// TwinCAT 3 PLC project STN500
// Title: STN500
// Company: Högskolan Väst
// Author: ANI
// ProgramVersion: 3.1.4022.3
// libraries:
//   Tc2_MC2, * (Beckhoff Automation GmbH)
//   Tc2_Standard, * (Beckhoff Automation GmbH)
//   Tc2_System, * (Beckhoff Automation GmbH)
//   Tc3_Module, * (Beckhoff Automation GmbH)
//   VisuDialogs, * (System)
//   VisuSymbols,3.5.10.0,System
// project tree:
//   DUTs/ AbsPosition.TcDUT, CommunicationData.TcDUT
//   / GlobalTextList.TcGTLO, PlcTask.TcTTO, Visualization Manager.TcVMO (not stored), VISU_TASK.TcTTO
//   GVLs/ GVL.TcGVL
//   POUs/ GantryPick.TcPOU, GantryLeave.TcPOU, GantryRobotMotion.TcPOU, GantryStatus.TcPOU, MAIN.TcPOU, PLC_PRG.TcPOU
//   VISUs/ GantryRobotVisu.TcVIS, Visualization.TcVIS
// real-time tasks:
//   TASK Device OPC UA Virtual Task: cycle T#200000us, priority 12, ADS port 350
//   TASK PlcTask: cycle T#5ms, priority 7, ADS port 351
//   TASK VISU_TASK: cycle T#100000us, priority 10, ADS port 352
// motion (NC):
//   TASK NC-Task 1 SAF: cycle T#2ms, priority 1, ADS port 501
//   TASK NC-Task 1 SVB: cycle T#4ms, priority 2, ADS port 511
//   AXIS Axis 1 (id 1)
//     General: UnitFlags=#x00000004
//     Dynamic: Acceleration=636.669, Deceleration=636.669, Jerk=445.433
//     Velo: Maximum=1000
//     OtherSettings: AllowMotionCmdToSlave=true
//     encoder EncType=19
//       EncPara: ScaleFactorNumerator=0.00162985, MaxCount=#xffffffff
//     drive DrvType=16
//       DrvPara: MaxCount=#xffffffff, DriveControlDWord=#x00020000
//         Analog: VeloReferenz=1000, ScaleFactorActTorque=0.1
//         TimeComp: TaskDelayCycles=1
//     controller CtrType=1
//       CtrPara: PriorControlFactor=1
//         PosDiffControl: Range=25
//         Observer: BandWidth=20
//   AXIS Axis 2 (id 2)
//     Dynamic: Acceleration=650.003, Deceleration=650.003, Jerk=444.737
//     Velo: Maximum=1000
//     OtherSettings: AllowMotionCmdToSlave=true
//     encoder EncType=19
//       EncPara: ScaleFactorNumerator=0.0005446764, MaxCount=#xffffffff
//     drive DrvType=16
//       DrvPara: MaxCount=#xffffffff, DriveControlDWord=#x00020000
//         Analog: VeloReferenz=1000, ScaleFactorActTorque=0.1
//         TimeComp: TaskDelayCycles=1
//     controller CtrType=1
//       CtrPara: PriorControlFactor=1
//         PosDiffControl: Range=25
//         Observer: BandWidth=20
//   AXIS Axis 3 (id 3)
//     Dynamic: Acceleration=630, Deceleration=630, Jerk=445.955
//     Velo: Maximum=1000
//     OtherSettings: AllowMotionCmdToSlave=true
//     encoder EncType=19
//       EncPara: ScaleFactorNumerator=0.000683214, MaxCount=#xffffffff
//     drive DrvType=16
//       DrvPara: MaxCount=#xffffffff, DriveControlDWord=#x00020000
//         Analog: VeloReferenz=1000, ScaleFactorActTorque=0.1
//         TimeComp: TaskDelayCycles=1
//     controller CtrType=1
//       CtrPara: PriorControlFactor=1
//         PosDiffControl: Range=25
//         Observer: BandWidth=20
// I/O:
//   DEVICE Device 1 (EtherCAT), AmsNetId 5.49.19.236.2.1
//     Term 1 (EK1200) PLC [EK1200-5000 EtherCAT Power supply (2A E-Bus)]
//       Term 2 (EK1110) [EK1110 EtherCAT extension]
//     Term 3 (EK1100) PLC Cabinet [EK1100 EtherCAT Coupler (2A E-Bus)]
//       Term 4 (EL1008) [EL1008 8Ch. Dig. Input 24V, 3ms]
//       Term 5 (EL1008) [EL1008 8Ch. Dig. Input 24V, 3ms]
//       Term 6 (EL2008) [EL2008 8Ch. Dig. Output 24V, 0.5A]
//       Term 7 (EL2008) [EL2008 8Ch. Dig. Output 24V, 0.5A]
//     Term 9 (EK1100) Gantry Robot Cabinet [EK1100 EtherCAT Coupler (2A E-Bus)]
//       Term 10 (EL1004) [EL1004 4Ch. Dig. Input 24V, 3ms]
//       Term 11 (EL1004) [EL1004 4Ch. Dig. Input 24V, 3ms]
//       Term 12 (EL1004) [EL1004 4Ch. Dig. Input 24V, 3ms]
//       Term 13 (EL2004) [EL2004 4Ch. Dig. Output 24V, 0.5A]
//       Term 16 (EL9011) [EL9011 End Terminal]
//     Drive X axis (MOVI-C MOVIDRIVE CiA402) [MOVI-C MOVIDRIVE CiA402]
//       modules: Module 1 (Mode of operation - CSP)
//     Drive Y Z axes (MOVI-C MOVIDRIVE CiA402) [MOVI-C MOVIDRIVE CiA402]
//       modules: Module 1 (Mode of operation - CSP), Module 3 (Mode of operation - CSP)
//   DEVICE Device 2 (OPC UA Virtual) STN100, AmsNetId 5.49.19.236.3.1
//   DEVICE Device 3 (OPC UA Virtual) STN200, AmsNetId 5.49.19.236.4.1
//   DEVICE Device 4 (OPC UA Virtual) STN300, AmsNetId 5.49.19.236.5.1
//   DEVICE Device 5 (OPC UA Virtual) STN400, AmsNetId 5.49.19.236.6.1
// variable links:
//   NC-Task 1 SAF/Axes/Axis 1 <-> Device 1 (EtherCAT)/Drive X axis (MOVI-C MOVIDRIVE CiA402)
//     Drive/Inputs/In/nDcOutputTime <-> InfoData/DcOutputShift
//     Drive/Inputs/In/nState1 <-> Module 1 (Mode of operation - CSP)/Inputs/Status word
//     Drive/Inputs/In/nState2 <-> Module 1 (Mode of operation - CSP)/Inputs/Status word @bit 8
//     Drive/Inputs/In/nState4 @bit 1 <-> WcState/InputToggle
//     Drive/Inputs/In/nState4 <-> WcState/WcState
//     Drive/Outputs/Out/nCtrl1 <-> Module 1 (Mode of operation - CSP)/Outputs/Control word
//     Drive/Outputs/Out/nCtrl2 <-> Module 1 (Mode of operation - CSP)/Outputs/Control word @bit 8
//     Drive/Outputs/Out/nDataOut1 <-> Module 1 (Mode of operation - CSP)/Outputs/Target position
//     Enc/Inputs/In/nDataIn1 <-> Module 1 (Mode of operation - CSP)/Inputs/Position actual value
//     Enc/Inputs/In/nDcInputTime <-> InfoData/DcInputShift
//     Enc/Inputs/In/nState4 @bit 1 <-> WcState/InputToggle
//     Enc/Inputs/In/nState4 <-> WcState/WcState
//   NC-Task 1 SAF/Axes/Axis 2 <-> Device 1 (EtherCAT)/Drive Y Z axes (MOVI-C MOVIDRIVE CiA402)
//     Drive/Inputs/In/nDcOutputTime <-> InfoData/DcOutputShift
//     Drive/Inputs/In/nState1 <-> Module 1 (Mode of operation - CSP)/Inputs/Status word
//     Drive/Inputs/In/nState2 <-> Module 1 (Mode of operation - CSP)/Inputs/Status word @bit 8
//     Drive/Inputs/In/nState4 @bit 1 <-> WcState/InputToggle
//     Drive/Inputs/In/nState4 <-> WcState/WcState
//     Drive/Outputs/Out/nCtrl1 <-> Module 1 (Mode of operation - CSP)/Outputs/Control word
//     Drive/Outputs/Out/nCtrl2 <-> Module 1 (Mode of operation - CSP)/Outputs/Control word @bit 8
//     Drive/Outputs/Out/nDataOut1 <-> Module 1 (Mode of operation - CSP)/Outputs/Target position
//     Enc/Inputs/In/nDataIn1 <-> Module 1 (Mode of operation - CSP)/Inputs/Position actual value
//     Enc/Inputs/In/nDcInputTime <-> InfoData/DcInputShift
//     Enc/Inputs/In/nState4 @bit 1 <-> WcState/InputToggle
//     Enc/Inputs/In/nState4 <-> WcState/WcState
//   NC-Task 1 SAF/Axes/Axis 3 <-> Device 1 (EtherCAT)/Drive Y Z axes (MOVI-C MOVIDRIVE CiA402)
//     Drive/Inputs/In/nDcOutputTime <-> InfoData/DcOutputShift
//     Drive/Inputs/In/nState1 <-> Module 3 (Mode of operation - CSP)/Inputs/Status word
//     Drive/Inputs/In/nState2 <-> Module 3 (Mode of operation - CSP)/Inputs/Status word @bit 8
//     Drive/Inputs/In/nState4 @bit 1 <-> WcState/InputToggle
//     Drive/Inputs/In/nState4 <-> WcState/WcState
//     Drive/Outputs/Out/nCtrl1 <-> Module 3 (Mode of operation - CSP)/Outputs/Control word
//     Drive/Outputs/Out/nCtrl2 <-> Module 3 (Mode of operation - CSP)/Outputs/Control word @bit 8
//     Drive/Outputs/Out/nDataOut1 <-> Module 3 (Mode of operation - CSP)/Outputs/Target position
//     Enc/Inputs/In/nDataIn1 <-> Module 3 (Mode of operation - CSP)/Inputs/Position actual value
//     Enc/Inputs/In/nDataIn6 @bit 1 <-> WcState/InputToggle
//     Enc/Inputs/In/nDataIn6 <-> WcState/WcState
//     Enc/Inputs/In/nDcInputTime <-> InfoData/DcInputShift
//   STN500/STN500 Instance <-> Device 1 (EtherCAT)/Term 3 (EK1100) PLC Cabinet/Term 4 (EL1008)
//     PlcTask Inputs/GVL.ixBtnControlOn <-> Channel 3/Input
//     PlcTask Inputs/GVL.ixBtnProgramStart <-> Channel 4/Input
//     PlcTask Inputs/GVL.ixBtnProgramStop <-> Channel 5/Input
//     PlcTask Inputs/GVL.ixEmergencyStopOk <-> Channel 1/Input
//     PlcTask Inputs/GVL.ixLightBeamAndGatesClosed <-> Channel 2/Input
//   STN500/STN500 Instance <-> Device 1 (EtherCAT)/Term 3 (EK1100) PLC Cabinet/Term 6 (EL2008)
//     PlcTask Outputs/GVL.qxIndControlOn <-> Channel 1/Output
//     PlcTask Outputs/GVL.qxIndProgramStart <-> Channel 2/Output
//     PlcTask Outputs/GVL.qxIndProgramStop <-> Channel 3/Output
//   STN500/STN500 Instance <-> Device 1 (EtherCAT)/Term 9 (EK1100) Gantry Robot Cabinet/Term 10 (EL1004)
//     PlcTask Inputs/GVL.ixCalSwY <-> Channel 2/Input
//     PlcTask Inputs/GVL.ixLimSwYNeg <-> Channel 3/Input
//     PlcTask Inputs/GVL.ixLimSwYPos <-> Channel 1/Input
//     PlcTask Inputs/GVL.ixLimSwZPos <-> Channel 4/Input
//   STN500/STN500 Instance <-> Device 1 (EtherCAT)/Term 9 (EK1100) Gantry Robot Cabinet/Term 11 (EL1004)
//     PlcTask Inputs/GVL.ixCalSwX <-> Channel 4/Input
//     PlcTask Inputs/GVL.ixCalSwZ <-> Channel 1/Input
//     PlcTask Inputs/GVL.ixLimSwX <-> Channel 3/Input
//     PlcTask Inputs/GVL.ixLimSwZNeg <-> Channel 2/Input
//   STN500/STN500 Instance <-> Device 1 (EtherCAT)/Term 9 (EK1100) Gantry Robot Cabinet/Term 13 (EL2004)
//     PlcTask Outputs/GVL.qxEnableSEWdrives <-> Channel 2/Output
//     PlcTask Outputs/GVL.qxGripper <-> Channel 1/Output
//   STN500/STN500 Instance <-> Device 2 (OPC UA Virtual) STN100/Object1 (OPC UA Client)/PLC1/GVL/iFromSTN500ToSTN100
//     PlcTask Outputs/GVL.iFromSTN500ToSTN100 <-> Outputs/Value
//   STN500/STN500 Instance <-> Device 2 (OPC UA Virtual) STN100/Object1 (OPC UA Client)/PLC1/GVL/iToSTN500FromSTN100
//     PlcTask Inputs/GVL.iToSTN500FromSTN100 <-> Inputs/Value
//   STN500/STN500 Instance <-> Device 3 (OPC UA Virtual) STN200/Object1 (OPC UA Client)/PLC1/GVL/iFromSTN500ToSTN200
//     PlcTask Outputs/GVL.iFromSTN500ToSTN200 <-> Outputs/Value
//   STN500/STN500 Instance <-> Device 3 (OPC UA Virtual) STN200/Object1 (OPC UA Client)/PLC1/GVL/iToSTN500FromSTN200
//     PlcTask Inputs/GVL.iToSTN500FromSTN200 <-> Inputs/Value
//   STN500/STN500 Instance <-> Device 4 (OPC UA Virtual) STN300/Object1 (OPC UA Client)/PLC1/GVL/iFromSTN500ToSTN300
//     PlcTask Outputs/GVL.iFromSTN500ToSTN300 <-> Outputs/Value
//   STN500/STN500 Instance <-> Device 4 (OPC UA Virtual) STN300/Object1 (OPC UA Client)/PLC1/GVL/iToSTN500FromSTN300
//     PlcTask Inputs/GVL.iToSTN500FromSTN300 <-> Inputs/Value
//   STN500/STN500 Instance <-> Device 5 (OPC UA Virtual) STN400/Object1 (OPC UA Client)/PLC1/GVL/iFromSTN500ToSTN400
//     PlcTask Outputs/GVL.iFromSTN500ToSTN400 <-> Outputs/Value
//   STN500/STN500 Instance <-> Device 5 (OPC UA Virtual) STN400/Object1 (OPC UA Client)/PLC1/GVL/iToSTN500FromSTN400
//     PlcTask Inputs/GVL.iToSTN500FromSTN400 <-> Inputs/Value
//   STN500/STN500 Instance <-> NC-Task 1 SAF/Axes/Axis 1
//     PlcTask Inputs/GantryRobotMotion.MCXAxisRef.NcToPlc <-> Outputs/ToPlc
//     PlcTask Outputs/GantryRobotMotion.MCXAxisRef.PlcToNc <-> Inputs/FromPlc
//   STN500/STN500 Instance <-> NC-Task 1 SAF/Axes/Axis 2
//     PlcTask Inputs/GantryRobotMotion.MCYAxisRef.NcToPlc <-> Outputs/ToPlc
//     PlcTask Outputs/GantryRobotMotion.MCYAxisRef.PlcToNc <-> Inputs/FromPlc
//   STN500/STN500 Instance <-> NC-Task 1 SAF/Axes/Axis 3
//     PlcTask Inputs/GantryRobotMotion.MCZAxisRef.NcToPlc <-> Outputs/ToPlc
//     PlcTask Outputs/GantryRobotMotion.MCZAxisRef.PlcToNc <-> Inputs/FromPlc

CONFIGURATION STN500
    RESOURCE PLC ON TwinCAT3
        TASK PlcTask(INTERVAL := T#5ms, PRIORITY := 7);
        TASK VISU_TASK(INTERVAL := T#100000us, PRIORITY := 10);
        PROGRAM MAIN WITH PlcTask : MAIN;
        PROGRAM VisuElems_Visu_Prg WITH VISU_TASK : VisuElems.Visu_Prg;
    END_RESOURCE
END_CONFIGURATION

// ---- DUTs/AbsPosition.TcDUT
TYPE AbsPosition :
STRUCT
	x:LREAL;
	y:LREAL;
	z:LREAL;
END_STRUCT
END_TYPE

// ---- DUTs/CommunicationData.TcDUT
TYPE CommunicationData :
STRUCT
	PickStation:INT;
	PickPosition:INT;
	AckPickStation:INT;
	AckPickPosition:INT;
	LeaveStation:INT;
	LeavePosition:INT;
	AckLeaveStation:INT;
	AckLeavePosition:INT;
	Status: STRING;
	ManualMode: BOOL;
	Auto: BOOL;
	Paus: BOOL;
END_STRUCT
END_TYPE

// ---- GVLs/GVL.TcGVL
{attribute 'qualified_only'}
VAR_GLOBAL
			
	//OPC-UA Communication
	iToSTN500FromSTN100 AT %I*: ARRAY[1..8] OF INT;		// From STN100
	iFromSTN500ToSTN100 AT %Q*: ARRAY[1..8] OF INT;		// To STN100

	iToSTN500FromSTN200 AT %I*: ARRAY[1..8] OF INT;		// From STN200
	iFromSTN500ToSTN200 AT %Q*: ARRAY[1..8] OF INT;		// To STN200

	iToSTN500FromSTN300 AT %I*: ARRAY[1..8] OF INT;		// From STN300
	iFromSTN500ToSTN300 AT %Q*: ARRAY[1..8] OF INT;		// To STN300

	
	iToSTN500FromSTN400 AT %I*: ARRAY[1..8] OF INT;		// From STN300
	iFromSTN500ToSTN400 AT %Q*: ARRAY[1..8] OF INT;		// To STN300
	

	//Digital I/O Gantry Robot	
	ixEmergencyStopOk		 	AT %I* 	: BOOL;			//Emergency stop reseted
	ixLightBeamAndGatesClosed 	AT %I* 	: BOOL;			//Gate closed and reseted
	ixBtnControlOn				AT %I*	: BOOL; 		//Button "Drift Till"
	ixBtnProgramStart			AT %I*	: BOOL;			//Button "Program Start"
	ixBtnProgramStop			AT %I*	: BOOL;			//Button "Program Stopp"

	ixLimSwYPos					AT %I*	: BOOL;			//End limit switches and calibration sensors
	ixCalSwY					AT %I*	: BOOL;
	ixLimSwYNeg					AT %I*	: BOOL;
	ixLimSwZPos					AT %I*	: BOOL;
	ixCalSwZ					AT %I*	: BOOL;
	ixLimSwZNeg					AT %I*	: BOOL;
	ixLimSwX					AT %I*	: BOOL;
	ixCalSwX					AT %I*	: BOOL;
	
	
	qxIndControlOn				AT %Q*	: BOOL; 		//Indication Lamp "Drift Till"
	qxIndProgramStart			AT %Q*	: BOOL;			//Indication Lamp Button "Program Start"
	qxIndProgramStop			AT %Q*	: BOOL;			//Indication Lamp Button "Program Stopp"

	qxGripper					AT %Q*	: BOOL;   		//Gripper pallets gantry robot
	qxEnableSEWdrives			AT %Q*  : BOOL;			//Enable motors XYZ axes
	
	ComData: CommunicationData;
	
END_VAR

// ---- POUs/MAIN.TcPOU
PROGRAM MAIN
VAR

END_VAR


GantryRobotMotion();
PLC_PRG();

END_PROGRAM

// ---- POUs/GantryRobotMotion.TcPOU
PROGRAM GantryRobotMotion
VAR
	
	//Speed settings Adjustible from Visu
	MCJogVelocity		: LREAL := 100.0;
	MCAutoVelocity		: LREAL := 250.0;
	mxMCButtonManLowVelocity 	: BOOL;
	

	//Homing motion Settings
	MCHomingMode	: MC_HomingMode := MC_HomingMode.MC_DefaultHoming ;
	iMCXCaibratePos 	: INT := 8;
	iMCYCaibratePos 	: INT := 8;
	iMCZCaibratePos 	: INT := 8;

	//Manual motion Settings
	MCJogMode		: E_JogMode 	:= E_JogMode.MC_JOGMODE_CONTINOUS;
	MCJogAcceleration	: LREAL := 500.0;
	MCJogDeceleration	: LREAL := 1500.0;
	MCJogJerk			: LREAL := 800.0;
	
	//Auto Motion Settings
	MCAutoAcceleration	: LREAL := 500.0;
	MCAutoDeceleration	: LREAL := 500.0;
	MCAutoJerk			: LREAL := 500.0;
	
	
	//Safe Transport Position
	MCYSafePos : LREAL := 160.0;
	MCZLiftDist : LREAL := 50.0;


	//Connection NC to Physical Servo Drives
	MCXAxisRef: AXIS_REF;
	MCYAxisRef: AXIS_REF;
	MCZAxisRef: AXIS_REF;

	
	// Auto motion Settings
	MCBufferMode   	: MC_BufferMode := MC_BufferMode.MC_Aborting;	
	
	

	//General Condition flags
	mxGeneralCOntrolOk: BOOL;
	mxButtonGeneralControlOn: BOOL;
	mxButtonGeneralControlOff: BOOL;
	mxButtonStartAuto : BOOL;
	mxButtonStopAuto : BOOL;
	mxButtonAutoMode: BOOL;
	mxGeneralControlOn: BOOL;	
	mxManualMode: BOOL;	
	mxAutoMode: BOOL;
	mxLimSwOK: BOOL;
	mxMCPowerOn: BOOL;
	mxAxesStatusOk: BOOL;
	mxAutoOn: BOOL;
	fbTONpuls1: TON;
	fbTONpuls2: TON;
	mxControlOff: BOOL;
	
	//Motor Control Function Block
	//MC  Power
	fbMCXPower: MC_Power;	//X-Axis
	mxMCXButtonByPass: BOOL;
	mxMCXPowerOn: BOOL;	

	fbMCYPower: MC_Power;	//Y-Axis
	mxMCYButtonByPass: BOOL;
	mxMCYPowerOn: BOOL;	
	
	fbMCZPower: MC_Power;	//Z-Axis
	mxMCZButtonByPass: BOOL;
	mxMCZPowerOn: BOOL;	
	
	
	// MC Read Status
	fbMCXReadStatus	: MC_ReadStatus;
	MCXAxisStatus	: ST_AxisStatus;
	mxMCXAxisError	: BOOL;

	fbMCYReadStatus	: MC_ReadStatus;
	MCYAxisStatus	: ST_AxisStatus;
	mxMCYAxisError	: BOOL;

	fbMCZReadStatus	: MC_ReadStatus;
	MCZAxisStatus	: ST_AxisStatus;
	mxMCZAxisError	: BOOL;

	
	// MC Read Actual Position
	fbMCXReadActualPosition: MC_ReadActualPosition;
	fbMCYReadActualPosition: MC_ReadActualPosition;
	fbMCZReadActualPosition: MC_ReadActualPosition;
	MCActualPos: AbsPosition;	
		
	//MC Reset
	fbMCXReset: MC_Reset;	
	fbMCYReset: MC_Reset;	
	fbMCZReset: MC_Reset;	
	mxButtonResetError:BOOL;

	//MC Homing 
	fbMCXHome: MC_Home;			//X-axis
	mxMCXButtonHoming: BOOL;
	mxMCXHomingDone: BOOL;	
	
	fbMCYHome: MC_Home;			//Y-axis
	mxMCYButtonHoming: BOOL;
	mxMCYHomingDone: BOOL;	
	
	fbMCZHome: MC_Home;			//Z-axis
	mxMCZButtonHoming: BOOL;
	mxMCZHomingDone: BOOL;	
	mxHomingDone: BOOL;	
	
	//MC Jog
	fbMCXJog: MC_Jog;			//X-Axis
	mxMCXButtonJogFWD: BOOL;
	mxMCXButtonJogBWD: BOOL;
	
	fbMCYJog: MC_Jog;			//Y-Axis
	mxMCYButtonJogFWD: BOOL;
	mxMCYButtonJogBWD: BOOL;
	
	fbMCZJog: MC_Jog;			//Z-Axis
	mxMCZButtonJogFWD: BOOL;
	mxMCZButtonJogBWD: BOOL;
	
	
	//MC Move Absolute Position	(Auto Sequence)
	fbMCXMoveAbsolute: MC_MoveAbsolute;		//X-Axis
	mxMCXMoveAbs: BOOL;
	MCXMovAbsPos: LREAL;
	MCXMoveAbsVel: LREAL;
	MCXMoveAbsACC: LREAL;
	MCXMoveAbsDec: LREAL;
	MCXMoveAbsJerk: LREAL;
	mxMCXMoveAbsDone: BOOL;

	//MC Move Absolute Position
	fbMCYMoveAbsolute: MC_MoveAbsolute;  	//Y-Axis
	mxMCYMoveAbs: BOOL;
	MCYMovAbsPos: LREAL;
	MCYMoveAbsVel: LREAL;
	MCYMoveAbsACC: LREAL;
	MCYMoveAbsDec: LREAL;
	MCYMoveAbsJerk: LREAL;
	mxMCYMoveAbsDone: BOOL;
	
	fbMCXHalt: MC_Halt;
	fbMCYHalt: MC_Halt;
	fbMCZHalt: MC_Halt;
	

	//MC Move Absolute Position
	fbMCZMoveAbsolute: MC_MoveAbsolute;		//Z-Axis
	mxMCZMoveAbs: BOOL;
	MCZMovAbsPos: LREAL;
	MCZMoveAbsVel: LREAL;
	MCZMoveAbsACC: LREAL;
	MCZMoveAbsDec: LREAL;
	MCZMoveAbsJerk: LREAL;
	mxMCZMoveAbsDone: BOOL;
	
	//Modify Position
	ModPos	: AbsPosition;
	ModPosStation: INT := 1;
	ModPosLocation:INT := 1;
	mxButtonModPosExecute : BOOL;
	mxButtonSavePos : BOOL;
	fbTONButtonModPosExecute : TON;
	mxButtonReadFile: BOOL;
	mxReminderToSave : BOOL;
	
	
	// Gripper	
	mxTogleGripper : BOOL;
	fbTONGripperOn: TON;
	fbTONGripperOff: TON;	
	
	//Auto Sequence
	iSequence: INT; 
	arrAbsPosition: ARRAY[1..4, 1..9] OF AbsPosition;	//Station 100-400 Place 1 to 9
	mxButtonGoToModPos : BOOL;
	strStatusText : STRING;
	
	
	//File handling AbsPositions XYZ
	fbFileOpen    			: FB_FileOpen;
    fbFileRead              : FB_FileRead;
    fbFileWrite             : FB_FileWrite;
    fbFileClose             : FB_FileClose;    
	hFile                   : UINT   := 0;
	mxFileOpen				: BOOL;
	mxFileRead				: BOOL;	
	mxFileWrite				: BOOL;
	mxFileClose				: BOOL;
	nFileOpenMode			: DWORD;
	mxMemSavePos: BOOL;
	mxMemReadFile: BOOL;
	fbTONFileTime: TON;

END_VAR
VAR // added by the converter: edge detectors and wires of the graphical bodies
    _rt1, _rt2, _rt3, _rt4, _rt5, _rt6, _rt7 : R_TRIG;
END_VAR

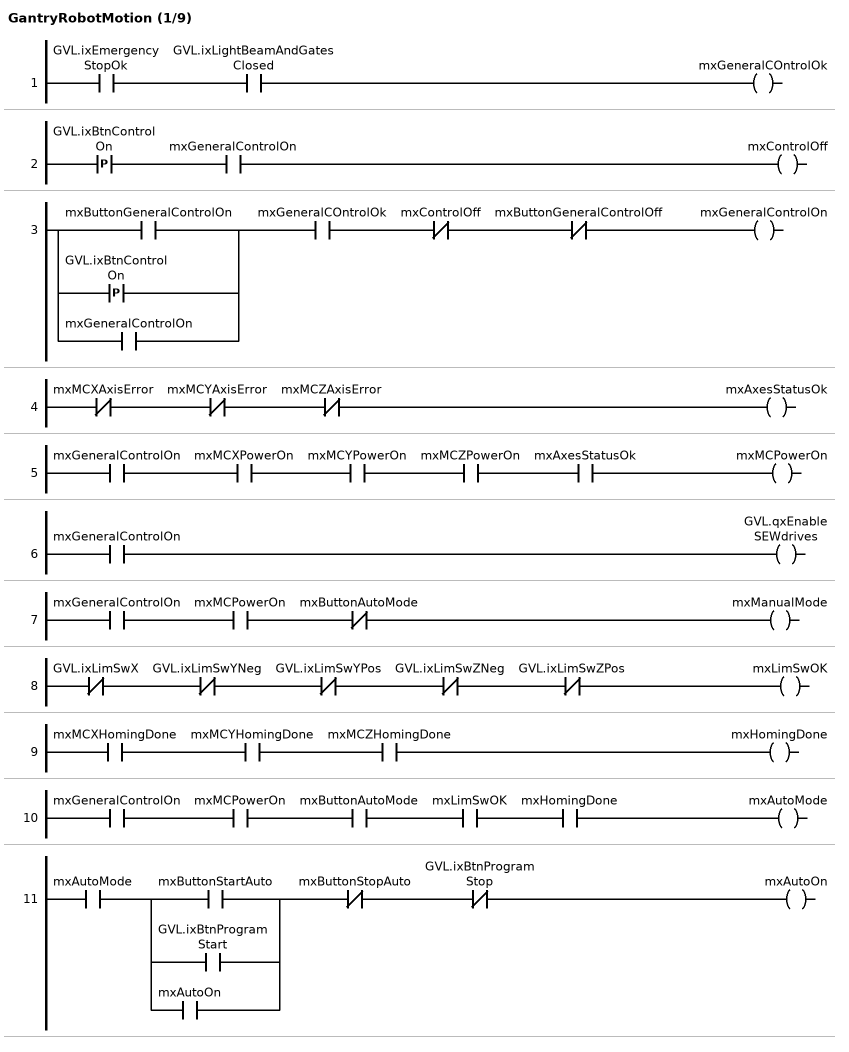
// NETWORK 1
mxGeneralCOntrolOk := GVL.ixEmergencyStopOk AND GVL.ixLightBeamAndGatesClosed;

// NETWORK 2
_rt1(CLK := GVL.ixBtnControlOn);
mxControlOff := _rt1.Q AND mxGeneralControlOn;

// NETWORK 3
_rt2(CLK := GVL.ixBtnControlOn);
mxGeneralControlOn := (mxButtonGeneralControlOn OR _rt2.Q OR mxGeneralControlOn) AND mxGeneralCOntrolOk AND NOT mxControlOff AND NOT mxButtonGeneralControlOff;

// NETWORK 4
mxAxesStatusOk := NOT mxMCXAxisError AND NOT mxMCYAxisError AND NOT mxMCZAxisError;

// NETWORK 5
mxMCPowerOn := mxGeneralControlOn AND mxMCXPowerOn AND mxMCYPowerOn AND mxMCZPowerOn AND mxAxesStatusOk;

// NETWORK 6
GVL.qxEnableSEWdrives := mxGeneralControlOn;

// NETWORK 7
mxManualMode := mxGeneralControlOn AND mxMCPowerOn AND NOT mxButtonAutoMode;

// NETWORK 8
mxLimSwOK := NOT GVL.ixLimSwX AND NOT GVL.ixLimSwYNeg AND NOT GVL.ixLimSwYPos AND NOT GVL.ixLimSwZNeg AND NOT GVL.ixLimSwZPos;

// NETWORK 9
mxHomingDone := mxMCXHomingDone AND mxMCYHomingDone AND mxMCZHomingDone;

// NETWORK 10
mxAutoMode := mxGeneralControlOn AND mxMCPowerOn AND mxButtonAutoMode AND mxLimSwOK AND mxHomingDone;

// NETWORK 11
mxAutoOn := mxAutoMode AND (mxButtonStartAuto OR GVL.ixBtnProgramStart OR mxAutoOn) AND NOT mxButtonStopAuto AND NOT GVL.ixBtnProgramStop;

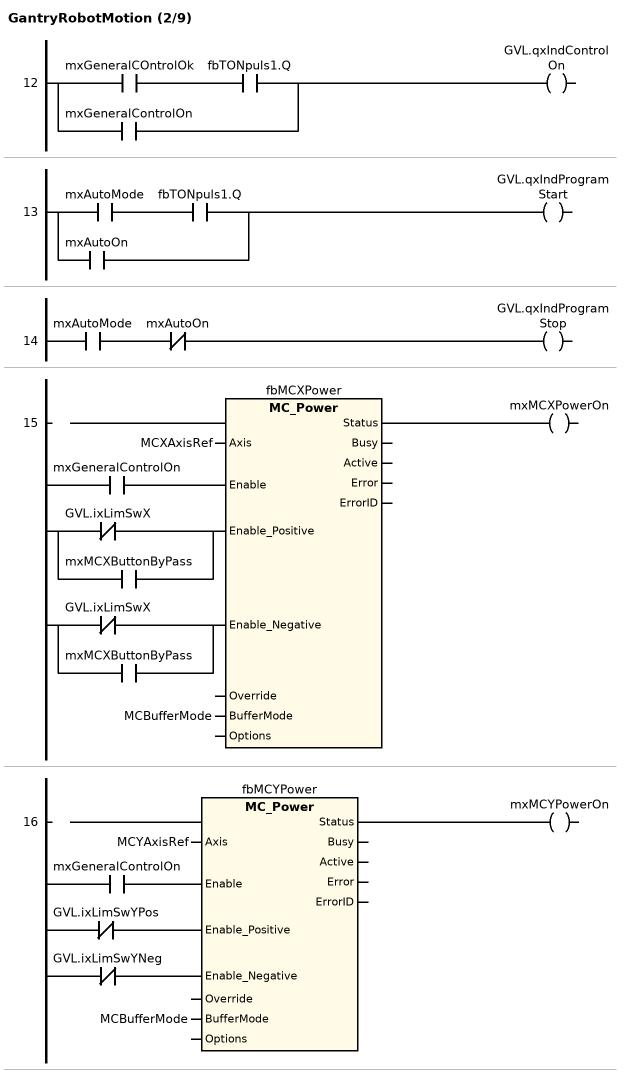
// NETWORK 12
GVL.qxIndControlOn := mxGeneralCOntrolOk AND fbTONpuls1.Q OR mxGeneralControlOn;

// NETWORK 13
GVL.qxIndProgramStart := mxAutoMode AND fbTONpuls1.Q OR mxAutoOn;

// NETWORK 14
GVL.qxIndProgramStop := mxAutoMode AND NOT mxAutoOn;

// NETWORK 15
fbMCXPower(
    Axis := MCXAxisRef,
    Enable := mxGeneralControlOn,
    Enable_Positive := NOT GVL.ixLimSwX OR mxMCXButtonByPass,
    Enable_Negative := NOT GVL.ixLimSwX OR mxMCXButtonByPass,
    BufferMode := MCBufferMode); // MC_Power
mxMCXPowerOn := fbMCXPower.Status;

// NETWORK 16
fbMCYPower(
    Axis := MCYAxisRef,
    Enable := mxGeneralControlOn,
    Enable_Positive := NOT GVL.ixLimSwYPos,
    Enable_Negative := NOT GVL.ixLimSwYNeg,
    BufferMode := MCBufferMode); // MC_Power
mxMCYPowerOn := fbMCYPower.Status;

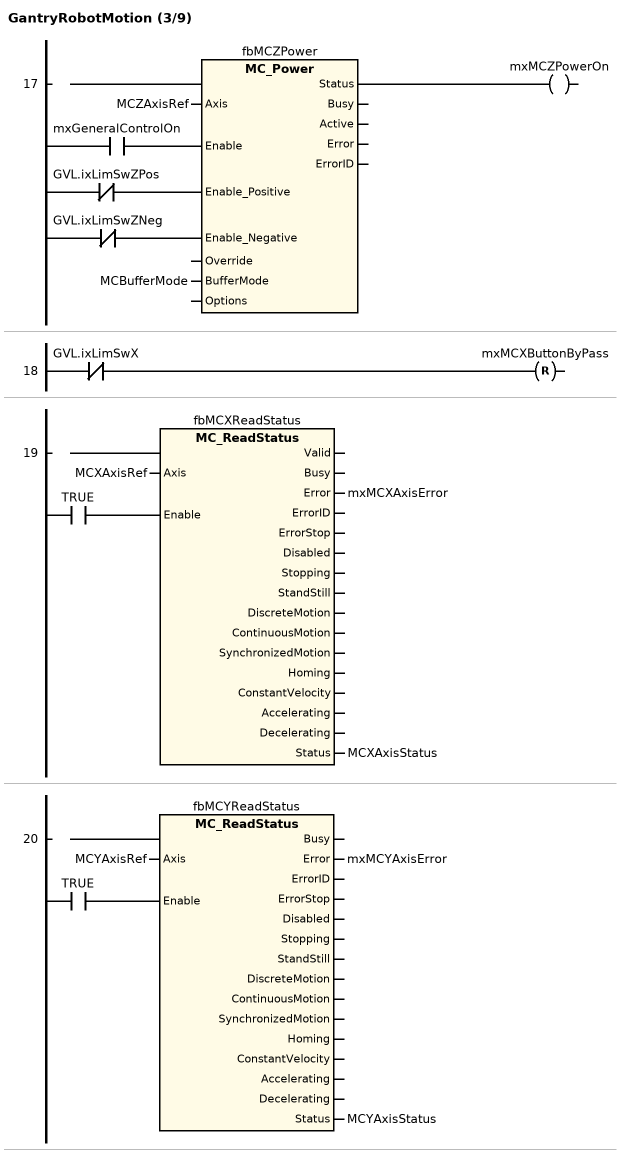
// NETWORK 17
fbMCZPower(
    Axis := MCZAxisRef,
    Enable := mxGeneralControlOn,
    Enable_Positive := NOT GVL.ixLimSwZPos,
    Enable_Negative := NOT GVL.ixLimSwZNeg,
    BufferMode := MCBufferMode); // MC_Power
mxMCZPowerOn := fbMCZPower.Status;

// NETWORK 18
mxMCXButtonByPass R= NOT GVL.ixLimSwX;

// NETWORK 19
fbMCXReadStatus(Axis := MCXAxisRef, Enable := TRUE, Error => mxMCXAxisError, Status => MCXAxisStatus); // MC_ReadStatus

// NETWORK 20
fbMCYReadStatus(Axis := MCYAxisRef, Enable := TRUE, Error => mxMCYAxisError, Status => MCYAxisStatus); // MC_ReadStatus

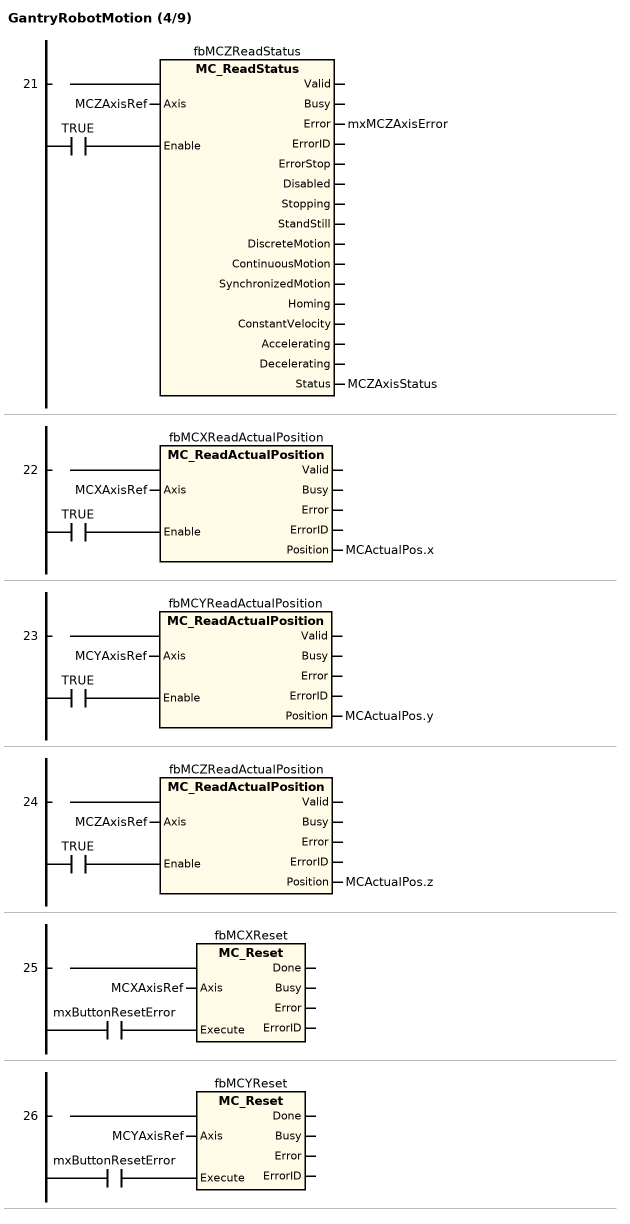
// NETWORK 21
fbMCZReadStatus(Axis := MCZAxisRef, Enable := TRUE, Error => mxMCZAxisError, Status => MCZAxisStatus); // MC_ReadStatus

// NETWORK 22
fbMCXReadActualPosition(Axis := MCXAxisRef, Enable := TRUE, Position => MCActualPos.x); // MC_ReadActualPosition

// NETWORK 23
fbMCYReadActualPosition(Axis := MCYAxisRef, Enable := TRUE, Position => MCActualPos.y); // MC_ReadActualPosition

// NETWORK 24
fbMCZReadActualPosition(Axis := MCZAxisRef, Enable := TRUE, Position => MCActualPos.z); // MC_ReadActualPosition

// NETWORK 25
fbMCXReset(Axis := MCXAxisRef, Execute := mxButtonResetError); // MC_Reset

// NETWORK 26
fbMCYReset(Axis := MCYAxisRef, Execute := mxButtonResetError); // MC_Reset

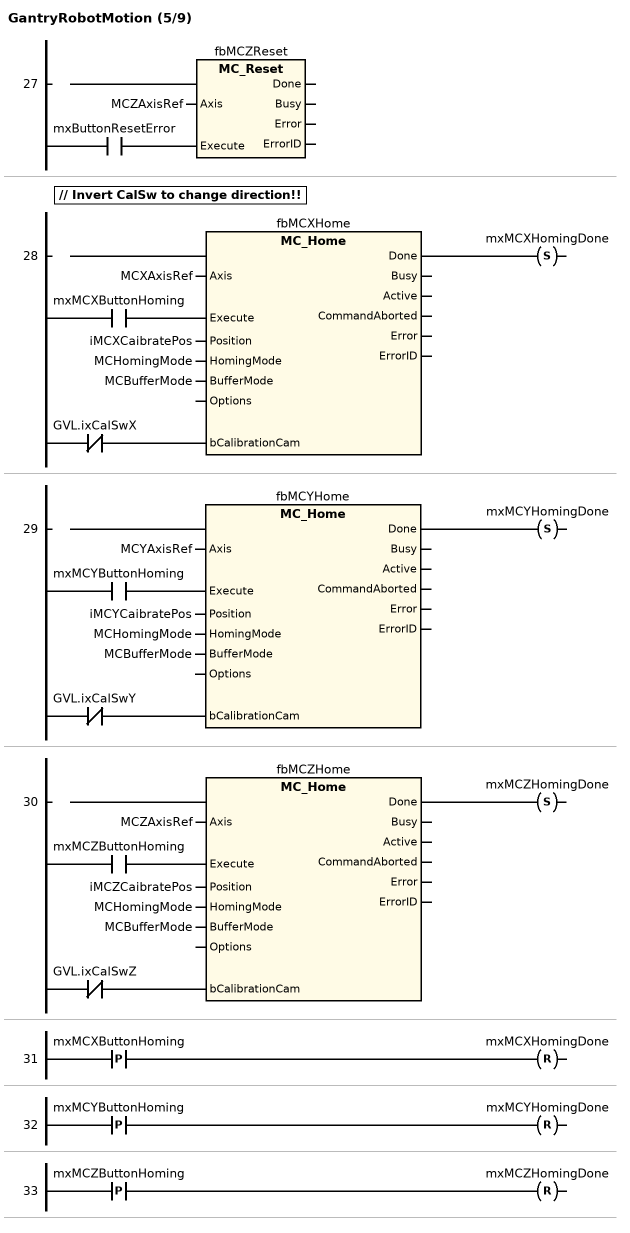
// NETWORK 27
fbMCZReset(Axis := MCZAxisRef, Execute := mxButtonResetError); // MC_Reset

// NETWORK 28
// label: // Invert CalSw to change direction!!
fbMCXHome(
    Axis := MCXAxisRef,
    Execute := mxMCXButtonHoming,
    Position := iMCXCaibratePos,
    HomingMode := MCHomingMode,
    BufferMode := MCBufferMode,
    bCalibrationCam := NOT GVL.ixCalSwX); // MC_Home
mxMCXHomingDone S= fbMCXHome.Done;

// NETWORK 29
fbMCYHome(
    Axis := MCYAxisRef,
    Execute := mxMCYButtonHoming,
    Position := iMCYCaibratePos,
    HomingMode := MCHomingMode,
    BufferMode := MCBufferMode,
    bCalibrationCam := NOT GVL.ixCalSwY); // MC_Home
mxMCYHomingDone S= fbMCYHome.Done;

// NETWORK 30
fbMCZHome(
    Axis := MCZAxisRef,
    Execute := mxMCZButtonHoming,
    Position := iMCZCaibratePos,
    HomingMode := MCHomingMode,
    BufferMode := MCBufferMode,
    bCalibrationCam := NOT GVL.ixCalSwZ); // MC_Home
mxMCZHomingDone S= fbMCZHome.Done;

// NETWORK 31
_rt3(CLK := mxMCXButtonHoming);
mxMCXHomingDone R= _rt3.Q;

// NETWORK 32
_rt4(CLK := mxMCYButtonHoming);
mxMCYHomingDone R= _rt4.Q;

// NETWORK 33
_rt5(CLK := mxMCZButtonHoming);
mxMCZHomingDone R= _rt5.Q;

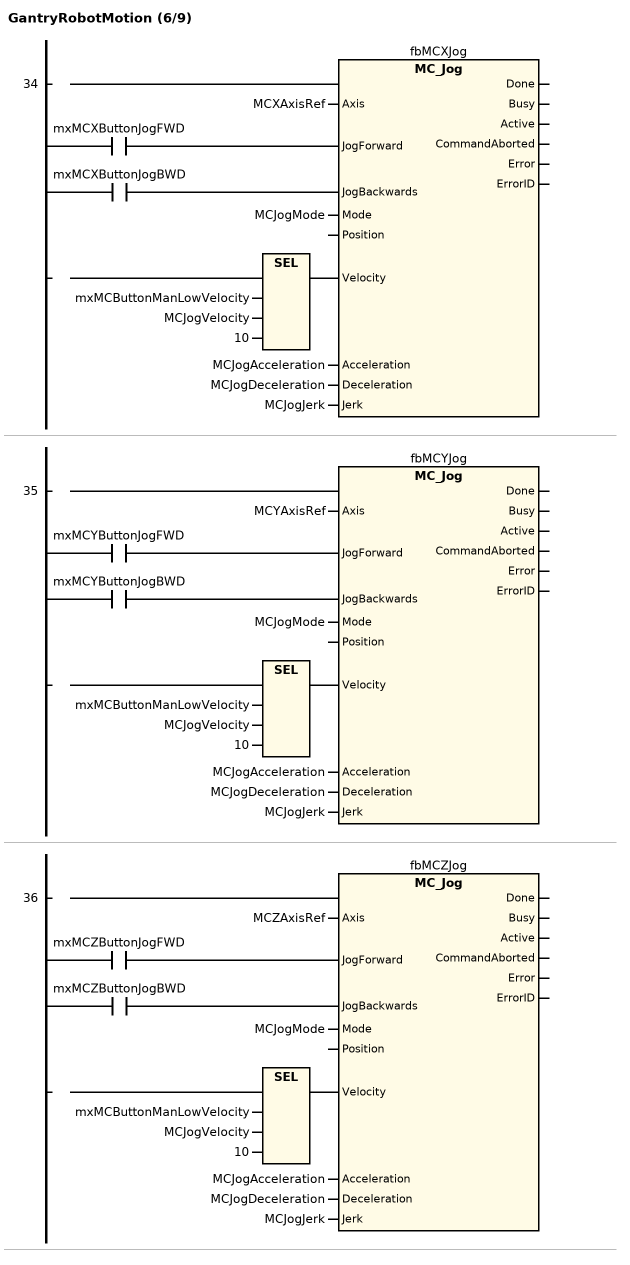
// NETWORK 34
fbMCXJog(
    Axis := MCXAxisRef,
    JogForward := mxMCXButtonJogFWD,
    JogBackwards := mxMCXButtonJogBWD,
    Mode := MCJogMode,
    Velocity := SEL(mxMCButtonManLowVelocity, MCJogVelocity, 10),
    Acceleration := MCJogAcceleration,
    Deceleration := MCJogDeceleration,
    Jerk := MCJogJerk); // MC_Jog

// NETWORK 35
fbMCYJog(
    Axis := MCYAxisRef,
    JogForward := mxMCYButtonJogFWD,
    JogBackwards := mxMCYButtonJogBWD,
    Mode := MCJogMode,
    Velocity := SEL(mxMCButtonManLowVelocity, MCJogVelocity, 10),
    Acceleration := MCJogAcceleration,
    Deceleration := MCJogDeceleration,
    Jerk := MCJogJerk); // MC_Jog

// NETWORK 36
fbMCZJog(
    Axis := MCZAxisRef,
    JogForward := mxMCZButtonJogFWD,
    JogBackwards := mxMCZButtonJogBWD,
    Mode := MCJogMode,
    Velocity := SEL(mxMCButtonManLowVelocity, MCJogVelocity, 10),
    Acceleration := MCJogAcceleration,
    Deceleration := MCJogDeceleration,
    Jerk := MCJogJerk); // MC_Jog

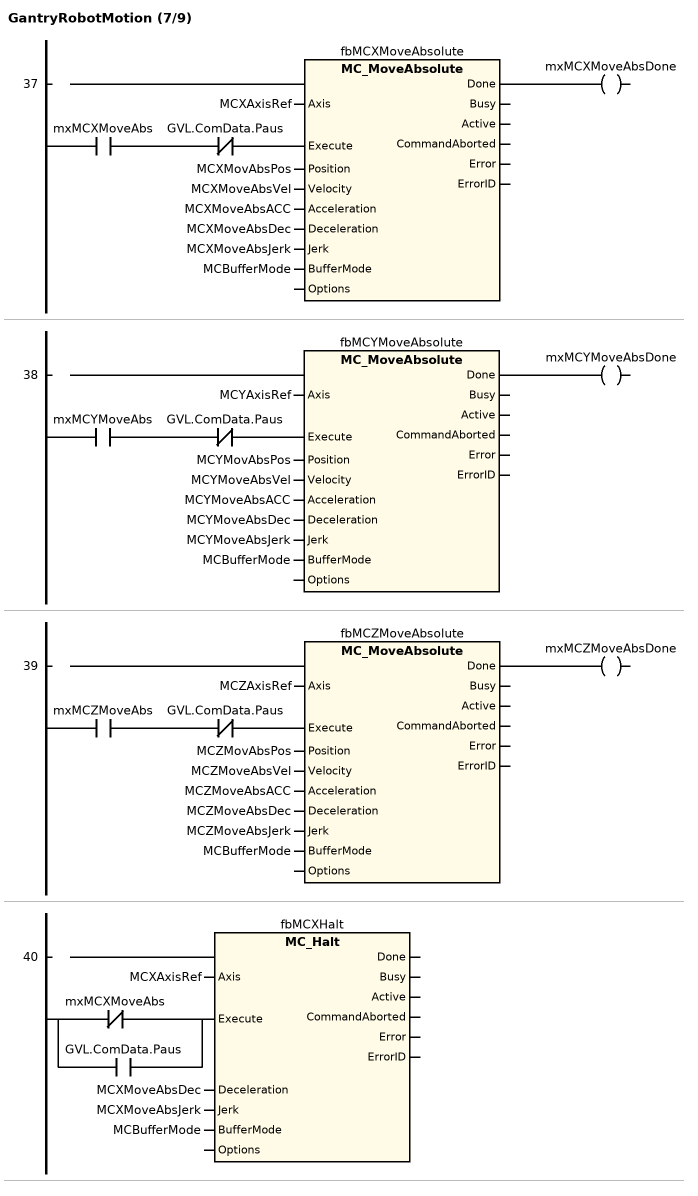
// NETWORK 37
fbMCXMoveAbsolute(
    Axis := MCXAxisRef,
    Execute := mxMCXMoveAbs AND NOT GVL.ComData.Paus,
    Position := MCXMovAbsPos,
    Velocity := MCXMoveAbsVel,
    Acceleration := MCXMoveAbsACC,
    Deceleration := MCXMoveAbsDec,
    Jerk := MCXMoveAbsJerk,
    BufferMode := MCBufferMode); // MC_MoveAbsolute
mxMCXMoveAbsDone := fbMCXMoveAbsolute.Done;

// NETWORK 38
fbMCYMoveAbsolute(
    Axis := MCYAxisRef,
    Execute := mxMCYMoveAbs AND NOT GVL.ComData.Paus,
    Position := MCYMovAbsPos,
    Velocity := MCYMoveAbsVel,
    Acceleration := MCYMoveAbsACC,
    Deceleration := MCYMoveAbsDec,
    Jerk := MCYMoveAbsJerk,
    BufferMode := MCBufferMode); // MC_MoveAbsolute
mxMCYMoveAbsDone := fbMCYMoveAbsolute.Done;

// NETWORK 39
fbMCZMoveAbsolute(
    Axis := MCZAxisRef,
    Execute := mxMCZMoveAbs AND NOT GVL.ComData.Paus,
    Position := MCZMovAbsPos,
    Velocity := MCZMoveAbsVel,
    Acceleration := MCZMoveAbsACC,
    Deceleration := MCZMoveAbsDec,
    Jerk := MCZMoveAbsJerk,
    BufferMode := MCBufferMode); // MC_MoveAbsolute
mxMCZMoveAbsDone := fbMCZMoveAbsolute.Done;

// NETWORK 40
fbMCXHalt(
    Axis := MCXAxisRef,
    Execute := NOT mxMCXMoveAbs OR GVL.ComData.Paus,
    Deceleration := MCXMoveAbsDec,
    Jerk := MCXMoveAbsJerk,
    BufferMode := MCBufferMode); // MC_Halt

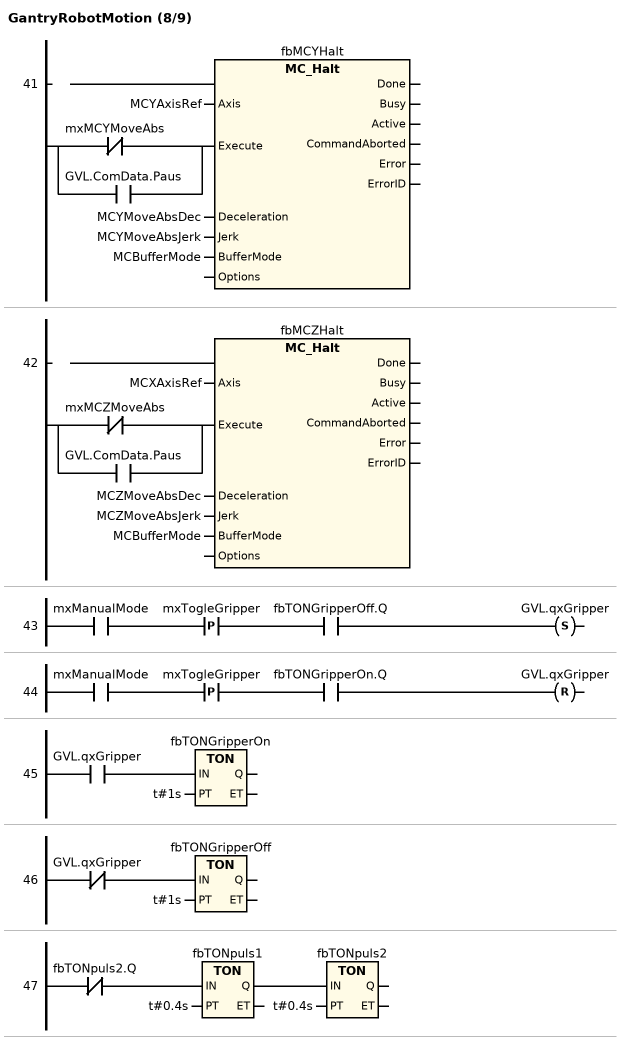
// NETWORK 41
fbMCYHalt(
    Axis := MCYAxisRef,
    Execute := NOT mxMCYMoveAbs OR GVL.ComData.Paus,
    Deceleration := MCYMoveAbsDec,
    Jerk := MCYMoveAbsJerk,
    BufferMode := MCBufferMode); // MC_Halt

// NETWORK 42
fbMCZHalt(
    Axis := MCXAxisRef,
    Execute := NOT mxMCZMoveAbs OR GVL.ComData.Paus,
    Deceleration := MCZMoveAbsDec,
    Jerk := MCZMoveAbsJerk,
    BufferMode := MCBufferMode); // MC_Halt

// NETWORK 43
_rt6(CLK := mxTogleGripper);
GVL.qxGripper S= mxManualMode AND _rt6.Q AND fbTONGripperOff.Q;

// NETWORK 44
_rt7(CLK := mxTogleGripper);
GVL.qxGripper R= mxManualMode AND _rt7.Q AND fbTONGripperOn.Q;

// NETWORK 45
fbTONGripperOn(IN := GVL.qxGripper, PT := t#1s); // TON

// NETWORK 46
fbTONGripperOff(IN := NOT GVL.qxGripper, PT := t#1s); // TON

// NETWORK 47
fbTONpuls1(IN := NOT fbTONpuls2.Q, PT := t#0.4s); // TON
fbTONpuls2(IN := fbTONpuls1.Q, PT := t#0.4s); // TON

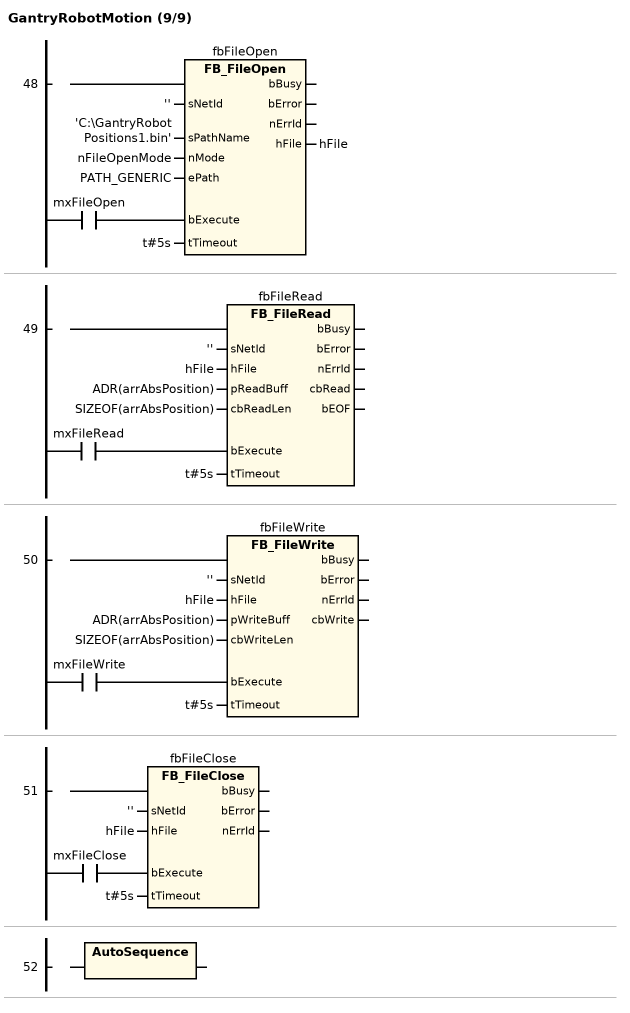
// NETWORK 48
fbFileOpen(
    sNetId := '',
    sPathName := 'C:\GantryRobotPositions1.bin',
    nMode := nFileOpenMode,
    ePath := PATH_GENERIC,
    bExecute := mxFileOpen,
    tTimeout := t#5s,
    hFile => hFile); // FB_FileOpen

// NETWORK 49
fbFileRead(
    sNetId := '',
    hFile := hFile,
    pReadBuff := ADR(arrAbsPosition),
    cbReadLen := SIZEOF(arrAbsPosition),
    bExecute := mxFileRead,
    tTimeout := t#5s); // FB_FileRead

// NETWORK 50
fbFileWrite(
    sNetId := '',
    hFile := hFile,
    pWriteBuff := ADR(arrAbsPosition),
    cbWriteLen := SIZEOF(arrAbsPosition),
    bExecute := mxFileWrite,
    tTimeout := t#5s); // FB_FileWrite

// NETWORK 51
fbFileClose(sNetId := '', hFile := hFile, bExecute := mxFileClose, tTimeout := t#5s); // FB_FileClose

// NETWORK 52
AutoSequence();

ACTION AutoSequence:


// Min Max Check Speed
IF MCJogVelocity > 250 THEN
	MCJogVelocity := 250;
END_IF
IF MCJogVelocity < 5 THEN
	MCJogVelocity := 5;
END_IF

IF MCAutoVelocity > 1000 THEN
	MCAutoVelocity := 1000;
END_IF
IF MCAutoVelocity < 100 THEN
	MCAutoVelocity := 100;
END_IF

	
// Copy status to function block interface
GVL.ComData.Status 		:= strStatusText;
GVL.ComData.ManualMode	:= mxManualMode;
GVL.ComData.Auto 		:= mxAutoOn;



CASE iSequence OF
	0:	// Init variable and read position file
		mxMCXMoveAbs := FALSE;
		mxMCYMoveAbs := FALSE;
		mxMCZMoveAbs := FALSE;
		fbTONButtonModPosExecute.PT := T#2S;
		fbTONButtonModPosExecute.IN := FALSE;
		fbTONButtonModPosExecute();

	
        // Open Gantry Robot Positions File for Read
		strStatusText := 'Reading Gantry Robot Position File'; 
		nFileOpenMode := FOPEN_MODEREAD OR FOPEN_MODEBINARY;
		mxFileOpen  := FALSE;
		mxFileRead  := FALSE;
		mxFileWrite := FALSE;
		mxFileClose := FALSE;	
		iSequence := 1;
		fbTONFileTime.IN := FALSE;
		fbTONFileTime.PT := T#3S;
		fbTONFileTime();
		
	
	1: // Wait for Opening of Gantry Robot Positions file and Check Errors
		fbTONFileTime.IN := TRUE;
		fbTONFileTime();
		mxFileOpen  := fbTONFileTime.q;
		IF mxFileOpen AND hFile > 0 AND NOT fbFileOpen.bBusy AND NOT fbFileOpen.bError THEN
			iSequence := 2;
		END_IF

	
	2:  // Read in Gantry Robot Positions File  to array of positions
		mxFileOpen  := FALSE;
		mxFileRead 	:= TRUE;
		iSequence := 3;		

			
	3:  // Wait for read Gantry Robot Positions File
		IF NOT fbFileRead.bBusy AND NOT fbFileRead.bError AND fbFileRead.cbRead = SIZEOF(arrAbsPosition) THEN
			iSequence := 4;
		END_IF
		

	4: // Close Gantry Robot Positions File
		mxFileRead  := FALSE;
		mxFileClose := TRUE;		
		strStatusText := 'Gantry Robot Position File Readed';		
		iSequence := 10;


	(* Write file *)
	5:  // Open Gantry Robot Positions Text File for Write
		strStatusText := 'Writing Gantry Robot Position File'; 
		nFileOpenMode := FOPEN_MODEWRITE OR FOPEN_MODEBINARY;
		mxFileOpen  := FALSE;
		mxFileRead  := FALSE;
		mxFileWrite := FALSE;
		mxFileClose := FALSE;	
		fbTONFileTime.IN := FALSE;
		fbTONFileTime.PT := T#3S;
		fbTONFileTime();
		iSequence := 6;
		
	
	6: // Wait for Opening of Gantry Robot Positions File and Check Errors
		fbTONFileTime.IN := TRUE;
		fbTONFileTime();
		mxFileOpen  := fbTONFileTime.Q;
		IF mxFileOpen AND hFile > 0 AND NOT fbFileOpen.bBusy AND NOT fbFileOpen.bError THEN
			iSequence := 7;
		END_IF
	
	
	7:  // Write Gantry Robot Positions File from array of positions
		mxFileOpen  := FALSE;
		mxFileWrite := TRUE;
		iSequence := 8;		

			
	8:	// Wait for Write Gantry Robot Positions File
		IF NOT fbFileWrite.bBusy AND NOT fbFileWrite.bError AND fbFileWrite.cbWrite = SIZEOF(arrAbsPosition) THEN
			iSequence := 9;
		END_IF


	9: 	// Close Gantry Robot Positions File
		strStatusText := 'Gantry Robot Positions Saved'; 		
		mxFileWrite  := FALSE;
		mxFileClose := TRUE;		
		iSequence := 10;

		
	10: // ********* Wait for auto or Modify Position, Save to file and status in Manual mode  ***************
	
		//Status text
		IF NOT GVL.ixEmergencyStopOk THEN
			strStatusText := 'Emergency Stop Activated';
		ELSIF NOT GVL.ixLightBeamAndGatesClosed THEN
			strStatusText := 'Safety Stop (Gate) Activated';
		ELSIF mxGeneralCOntrolOk AND NOT mxGeneralControlOn THEN
			strStatusText := 'Ready for General Power';
		ELSIF mxGeneralControlOn AND NOT mxMCPowerOn THEN
			strStatusText := 'Servo Drives Fault';
		ELSIF mxManualMode THEN
			strStatusText := 'Manual Mode OK';	
		ELSIF mxButtonAutoMode AND NOT mxLimSwOK THEN
			strStatusText := 'End Limit Switch Activated';
		ELSIF mxButtonAutoMode AND NOT mxHomingDone THEN
			strStatusText := 'Axes Not in reference (Run Homing)';
		ELSIF mxButtonAutoMode AND NOT mxAutoOn THEN
			strStatusText := 'Ready for Start Auto';
		ELSIF mxAutoOn THEN
			strStatusText := 'Ready for Order Auto';
		END_IF
		
					
		// Run in auto mode
		IF mxAutoOn THEN
			iSequence := 100;
		END_IF
	
		GVL.ComData.AckPickPosition := 0;
		GVL.ComData.AckPickStation := 0;
		GVL.ComData.AckLeavePosition := 0;
		GVL.ComData.AckLeaveStation := 0;
		
	
		// Move to "Modify Position" in HMI selected Robot Station and Storage Loacation 
		IF mxButtonGoToModPos AND mxManualMode AND mxHomingDone THEN //Manual Mode
			iSequence := 20;	
		END_IF
		
		// Modify position
		IF  mxButtonModPosExecute AND mxManualMode THEN
			arrAbsPosition[ModPosStation, ModPosLocation] := MCActualPos;
			mxReminderToSave := TRUE;
		END_IF
		
		// Save Position
		IF mxButtonSavePos AND NOT mxMemSavePos THEN
			iSequence := 5; //Write file
			mxReminderToSave := FALSE;
		END_IF
		mxMemSavePos := mxButtonSavePos;
		
		// Read file (UnDo)
		IF mxButtonReadFile AND NOT mxMemReadFile THEN
			iSequence := 0; //Read file
			mxReminderToSave := FALSE;
		END_IF
		mxMemReadFile := mxButtonReadFile;
		
		// Auto motion	
		IF mxAutoOn THEN
			IF GVL.ComData.LeavePosition = 0 
				AND GVL.ComData.LeaveStation = 0 
					AND GVL.ComData.PickPosition = 0 
						AND GVL.ComData.PickStation = 0 	THEN
				iSequence := 100;		//Auto mode					
			ELSE
				strStatusText := 'Clear Old Order';
			END_IF;
		END_IF
		

	
	20: 	//Init Speed Acc Dec Jerk for Manual Mode ( Goto ModPos) 
		MCXMoveAbsVel	:= MCJogVelocity ;
		MCXMoveAbsACC	:= MCJogAcceleration;
		MCXMoveAbsDec	:= MCJogDeceleration;
		MCXMoveAbsJerk	:= MCJogJerk;

		MCYMoveAbsVel	:= MCJogVelocity ;
		MCYMoveAbsACC	:= MCJogAcceleration;
		MCYMoveAbsDec	:= MCJogDeceleration;
		MCYMoveAbsJerk	:= MCJogJerk;

		MCZMoveAbsVel	:= MCJogVelocity ;
		MCZMoveAbsACC	:= MCJogAcceleration;
		MCZMoveAbsDec	:= MCJogDeceleration;
		MCZMoveAbsJerk	:= MCJogJerk;
		strStatusText := 'Moving to Modify Position';

		iSequence := 30;
		
		
	30:		// Move Y to safe position in the passage ( Goto ModPos)
		MCYMovAbsPos	:= MCYSafePos;
		mxMCYMoveAbs	:= TRUE;
		
		IF mxMCYMoveAbsDone THEN
			mxMCYMoveAbs := FALSE;
			iSequence := 40;
		END_IF
		
 		IF NOT mxButtonGoToModPos OR NOT mxManualMode THEN
			mxMCYMoveAbs:= FALSE;
			iSequence := 10;
		END_IF

		
	40:		// Move X And Z to Above Loacation ( Goto ModPos)
		MCXMovAbsPos	:= arrAbsPosition[ ModPosStation, ModPosLocation].x;
		mxMCXMoveAbs	:= TRUE;

		MCZMovAbsPos	:= arrAbsPosition[ ModPosStation, ModPosLocation].z - MCZLiftDist;
		mxMCZMoveAbs	:= TRUE;

	
		IF mxMCXMoveAbsDone AND mxMCZMoveAbsDone THEN
			mxMCXMoveAbs:= FALSE;
			mxMCZMoveAbs:= FALSE;
			iSequence 	:= 50;
		END_IF
		
		IF NOT mxButtonGoToModPos OR NOT mxManualMode THEN
			mxMCXMoveAbs:= FALSE;
			mxMCZMoveAbs:= FALSE;
			iSequence 	:= 10;
		END_IF
	
		
	50:		// Move Y in to storage ( Goto ModPos)
		MCYMovAbsPos		:= arrAbsPosition[ ModPosStation, ModPosLocation].y;
		mxMCYMoveAbs		:= TRUE;
		
		IF mxMCYMoveAbsDone THEN
			mxMCYMoveAbs 	:= FALSE;
			iSequence 		:= 60;
		END_IF
		
		IF NOT mxButtonGoToModPos OR NOT mxManualMode THEN
			mxMCYMoveAbs	:= FALSE;
			iSequence 		:= 0;
		END_IF
		
		
	60:		// Move Z down to storage ( Go to ModPos)	
		MCZMovAbsPos	:= arrAbsPosition[ ModPosStation, ModPosLocation].z;
		mxMCZMoveAbs	:= TRUE;
		
		IF mxMCYMoveAbsDone THEN
			strStatusText := 'In Modify Position';
		END_IF
		
		IF NOT mxButtonGoToModPos OR NOT mxManualMode THEN
			mxMCZMoveAbs:= FALSE;
			iSequence 	:= 10;
		END_IF

	
	
	100: 	// Init Auto speed acc and jerk ( Auto)
		MCXMoveAbsVel	:= MCAutoVelocity ;
		MCXMoveAbsACC	:= MCAutoAcceleration;
		MCXMoveAbsDec	:= MCAutoDeceleration;
		MCXMoveAbsJerk	:= MCAutoJerk;

		MCYMoveAbsVel	:= MCAutoVelocity ;
		MCYMoveAbsACC	:= MCAutoAcceleration;
		MCYMoveAbsDec	:= MCAutoDeceleration;
		MCYMoveAbsJerk	:= MCAutoJerk;

		MCZMoveAbsVel	:= MCAutoVelocity ;
		MCZMoveAbsACC	:= MCAutoAcceleration;
		MCZMoveAbsDec	:= MCAutoDeceleration;
		MCZMoveAbsJerk	:= MCAutoJerk;

		iSequence 		:= 110;

		
	110:  // Move Y to safe position in the passage ( Auto)
		MCYMovAbsPos	:= MCYSafePos;
		mxMCYMoveAbs	:= TRUE;
		strStatusText := 'Moving Y-axis to Transport Position';
	
		IF mxMCYMoveAbsDone THEN
			mxMCYMoveAbs := FALSE;
			iSequence := 120;
		END_IF
		
		IF NOT mxAutoOn THEN
			mxMCYMoveAbs:= FALSE;
			iSequence := 10;
		END_IF	

	
	120: 	// Ready for order  ( Auto)
		strStatusText := 'Ready for Order';
		iSequence := 130;

		IF NOT mxAutoOn THEN
			iSequence := 10;
		END_IF
		
		
	130:  	// *************************************** Wait for order ( Auto)  **************************************************
		IF GVL.ComData.PickPosition > 0	AND GVL.ComData.PickStation > 0 THEN
			GVL.ComData.AckPickPosition	:= 	GVL.ComData.PickPosition; //Acknowledge to function block
			GVL.ComData.AckPickStation	:= 	GVL.ComData.PickStation;
			iSequence := 200;
		END_IF		

		IF GVL.ComData.LeavePosition > 0 AND GVL.ComData.LeaveStation > 0 THEN
			GVL.ComData.AckLeavePosition	:= 	GVL.ComData.LeavePosition;
			GVL.ComData.AckLeaveStation		:= 	GVL.ComData.LeaveStation;
			iSequence := 300;
		END_IF
		

		IF NOT mxAutoOn THEN
			iSequence := 10;
		END_IF
		

	(* Auto Pickup sequence *)
	200: 	//Check Order (Auto Pickup) 	
		IF  GVL.ComData.PickPosition > 0 
			AND GVL.ComData.PickPosition <=9 
				AND GVL.ComData.PickStation > 0 
					AND GVL.ComData.PickStation <= 4 THEN
			iSequence := 210;
		ELSE
			strStatusText := 'Wrong Pickup Order Address';
			IF GVL.ComData.PickPosition = 0 AND GVL.ComData.PickStation = 0 THEN
				iSequence := 10;
			END_IF
		END_IF

		IF NOT mxAutoOn OR GVL.ComData.PickPosition = 0 OR	 GVL.ComData.PickStation = 0 THEN
			iSequence := 10;
		END_IF


	210:	// Move X And Z to Above and Outside the Loacation ( Auto Pickup)

		MCXMovAbsPos	:=  arrAbsPosition[ GVL.ComData.PickStation, GVL.ComData.PickPosition].x;
		mxMCXMoveAbs	:= TRUE;

		MCZMovAbsPos	:= arrAbsPosition[ GVL.ComData.PickStation, GVL.ComData.PickPosition].z - MCZLiftDist;
		mxMCZMoveAbs	:= TRUE;
		
		GVL.qxGripper := FALSE;
		strStatusText := 'Moving to Pickup Pallet';
		

		IF mxMCXMoveAbsDone AND mxMCZMoveAbsDone THEN
			mxMCXMoveAbs:= FALSE;
			mxMCZMoveAbs:= FALSE;
			iSequence 	:= 220;
		END_IF

		
		IF NOT mxAutoOn OR GVL.ComData.PickPosition = 0 OR	 GVL.ComData.PickStation = 0 THEN
			mxMCXMoveAbs:= FALSE;
			mxMCZMoveAbs:= FALSE;
			iSequence 	:= 10;
		END_IF
	
		
	220:	// Move Y in to storage (  Auto Pickup)
		MCYMovAbsPos		:=  arrAbsPosition[ GVL.ComData.PickStation, GVL.ComData.PickPosition].y;
		mxMCYMoveAbs		:= TRUE;
	
		IF mxMCYMoveAbsDone THEN
			mxMCYMoveAbs 	:= FALSE;
			iSequence 		:= 230;
		END_IF
		
		IF NOT mxAutoOn OR GVL.ComData.PickPosition = 0 OR	 GVL.ComData.PickStation = 0 THEN
			mxMCYMoveAbs	:= FALSE;
			iSequence 		:= 10;
		END_IF
			
		
	230:	// Move Z down to storage ( Auto Pickup)	
		MCZMovAbsPos	:= arrAbsPosition[ GVL.ComData.PickStation, GVL.ComData.PickPosition].z;
		mxMCZMoveAbs	:= TRUE;
		GVL.qxGripper := FALSE;
		
		IF mxMCZMoveAbsDone THEN
			mxMCZMoveAbs:= FALSE;
			iSequence 	:= 240;				
		END_IF
		
		IF NOT mxAutoOn OR GVL.ComData.PickPosition = 0 OR	 GVL.ComData.PickStation = 0  THEN
			mxMCZMoveAbs:= FALSE;
			iSequence 	:= 10;
		END_IF
		
	
	240:	//Grip pallet ( Auto Pickup)	
		GVL.qxGripper 	:= TRUE;
		strStatusText := 'Gripping the Pallet';
		IF fbTONGripperOn.Q THEN
			iSequence := 250;
		END_IF 
		
		IF NOT mxAutoOn OR GVL.ComData.PickPosition = 0 OR	 GVL.ComData.PickStation = 0  THEN
			iSequence 	:= 10;
		END_IF
		
		
	250: 	// Move Z up above storage ( Auto Pickup)	
		MCZMovAbsPos	:= arrAbsPosition[ GVL.ComData.PickStation, GVL.ComData.PickPosition].z - MCZLiftDist;
		mxMCZMoveAbs	:= TRUE;
		strStatusText := 'Moving out with the Pallet';
		
		IF mxMCZMoveAbsDone THEN
			mxMCZMoveAbs:= FALSE;
			iSequence := 260;
		END_IF
		
		IF NOT mxAutoOn OR GVL.ComData.PickPosition = 0 OR	 GVL.ComData.PickStation = 0  THEN
			mxMCZMoveAbs:= FALSE;
			iSequence 	:= 10;
		END_IF
		
		
	260:  	// Move Y to transport position ( Auto Pickup)	
		MCYMovAbsPos	:= MCYSafePos;
		mxMCYMoveAbs	:= TRUE;
	
		IF mxMCYMoveAbsDone THEN
			mxMCYMoveAbs := FALSE;
			GVL.ComData.AckPickPosition := 0;
			GVL.ComData.AckPickStation := 0;
			iSequence := 270;
		END_IF		
		
		IF NOT mxAutoOn OR GVL.ComData.PickPosition = 0 OR	 GVL.ComData.PickStation = 0 THEN
			mxMCYMoveAbs:= FALSE;
			iSequence := 10;
		END_IF

	
	270: 	// Wait for clear order
		strStatusText := 'Pickup pallet Done, Clear the order';
		IF 	GVL.ComData.PickStation = 0 AND GVL.ComData.PickPosition = 0 THEN
			strStatusText := 'Ready for Leave Order';
			iSequence := 130;
		END_IF	
		
		IF NOT mxAutoOn THEN
			mxMCYMoveAbs:= FALSE;
			iSequence := 10;
		END_IF

		
	300:  // Check Order 	( Auto Leave)
		IF  GVL.ComData.LeavePosition > 0 
			AND GVL.ComData.LeavePosition <=9 
				AND GVL.ComData.LeaveStation > 0 
					AND GVL.ComData.LeaveStation <= 4 THEN
			iSequence := 310;
		ELSE
			strStatusText := 'Wrong Leave Order Address';
			IF GVL.ComData.LeavePosition = 0 AND GVL.ComData.LeaveStation = 0 THEN
				iSequence := 10;
			END_IF
		END_IF

		IF NOT mxAutoOn THEN
			iSequence := 10;
		END_IF

	310:	// Move X And Z to Above and Outside the Loacation ( Auto Leave)
		MCXMovAbsPos	:= arrAbsPosition[ GVL.ComData.LeaveStation, GVL.ComData.LeavePosition].x;
		mxMCXMoveAbs	:= TRUE;

		MCZMovAbsPos	:= arrAbsPosition[ GVL.ComData.LeaveStation, GVL.ComData.LeavePosition].z - MCZLiftDist;
		mxMCZMoveAbs	:= TRUE;
		strStatusText := 'Moving to Leave Pallet';

		IF mxMCXMoveAbsDone AND mxMCZMoveAbsDone THEN
			mxMCXMoveAbs:= FALSE;
			mxMCZMoveAbs:= FALSE;
			iSequence 	:= 320;
		END_IF
		
		IF NOT mxAutoOn OR GVL.ComData.LeavePosition = 0 OR	 GVL.ComData.LeaveStation = 0 THEN
			mxMCXMoveAbs:= FALSE;
			mxMCZMoveAbs:= FALSE;
			iSequence 	:= 10;
		END_IF
	
		
	320:	// Move Y in to storage (  Auto Leave)
		MCYMovAbsPos		:= arrAbsPosition[ GVL.ComData.LeaveStation, GVL.ComData.LeavePosition].y;
		mxMCYMoveAbs		:= TRUE;
	
		IF mxMCYMoveAbsDone THEN
			mxMCYMoveAbs 	:= FALSE;
			iSequence 		:= 330;
		END_IF
		
		IF NOT mxAutoOn OR GVL.ComData.LeavePosition = 0 OR	 GVL.ComData.LeaveStation = 0 THEN
			mxMCYMoveAbs	:= FALSE;
			iSequence 		:= 10;
		END_IF
			
		
	330:	// Move Z down to storage ( Auto Leave)	
		MCZMovAbsPos	:= arrAbsPosition[ GVL.ComData.LeaveStation, GVL.ComData.LeavePosition].z;
		mxMCZMoveAbs	:= TRUE;
		
		IF mxMCZMoveAbsDone THEN
			mxMCZMoveAbs:= FALSE;
			iSequence 	:= 340;				
		END_IF
		
		IF NOT mxAutoOn OR GVL.ComData.LeavePosition = 0 OR	 GVL.ComData.LeaveStation = 0  THEN
			mxMCZMoveAbs:= FALSE;
			iSequence 	:= 10;
		END_IF
		
		
	340: 	// Release Gripper ( Auto Leave)
		GVL.qxGripper 	:= FALSE;
		strStatusText := 'Ungriping the Pallet';
		IF fbTONGripperOff.Q THEN
			iSequence := 350;
		END_IF 
		
		IF NOT mxAutoOn OR GVL.ComData.LeavePosition = 0 OR	 GVL.ComData.LeaveStation = 0  THEN
			iSequence 	:= 0;
		END_IF
		
		
	350:	// Move Z up above storage ( Auto Leave)	
		MCZMovAbsPos	:= arrAbsPosition[ GVL.ComData.LeaveStation, GVL.ComData.LeavePosition].z - MCZLiftDist;
		mxMCZMoveAbs	:= TRUE;
		strStatusText := 'Moving up from storage';
		
		IF mxMCZMoveAbsDone AND fbTONGripperOff.Q THEN
			mxMCZMoveAbs := FALSE;
			iSequence 	 := 360;
		END_IF
		
		IF NOT mxAutoOn OR GVL.ComData.LeavePosition = 0 OR	 GVL.ComData.LeaveStation = 0  THEN
			mxMCZMoveAbs := FALSE;
			iSequence 	 := 10;
		END_IF
		
		
	360: 	// Move Y to transport position ( Auto Leave)	
		MCYMovAbsPos	:= MCYSafePos;
		mxMCYMoveAbs	:= TRUE;
		strStatusText 	:= 'Moving out from storage';
	
		IF mxMCYMoveAbsDone THEN
			mxMCYMoveAbs := FALSE;
			GVL.ComData.AckLeavePosition := 0;
			GVL.ComData.AckLeaveStation := 0;
			iSequence 	 := 370;
		END_IF		
		
		IF NOT mxAutoOn OR GVL.ComData.LeavePosition = 0 OR	 GVL.ComData.LeaveStation = 0 THEN
			mxMCYMoveAbs:= FALSE;
			iSequence := 10;
		END_IF

		
	370: 	// Wait for clear order
		strStatusText 	:= 'Leave pallet Done, Clear the order';
		IF 	GVL.ComData.LeaveStation = 0 AND GVL.ComData.LeavePosition = 0 THEN
			strStatusText := 'Ready for Order';
			iSequence := 130;
		END_IF	
		
		IF NOT mxAutoOn THEN
			mxMCYMoveAbs:= FALSE;
			iSequence := 10;
		END_IF

	
END_CASE
END_ACTION

END_PROGRAM

// ---- POUs/PLC_PRG.TcPOU
PROGRAM PLC_PRG
VAR
	//Visualisation 	
	mxButtonPaus	: BOOL;

	mxAuto			: BOOL;

	//Internal use
	mxStart: BOOL;
	mxDone: BOOL;
	
	//Motion Function Blocks
	fbGantryStatus: GantryStatus;

	fbGantryPick_1: GantryPick;
	fbGantryLeave_2: GantryLeave;

	nPickStation: INT := 1;
	nPickPosition: INT := 1;
	nLeaveStation: INT := 1;
	nLeavePosition: INT := 2;
END_VAR
VAR // added by the converter: edge detectors and wires of the graphical bodies
    _w1, _w2 : BOOL;
END_VAR

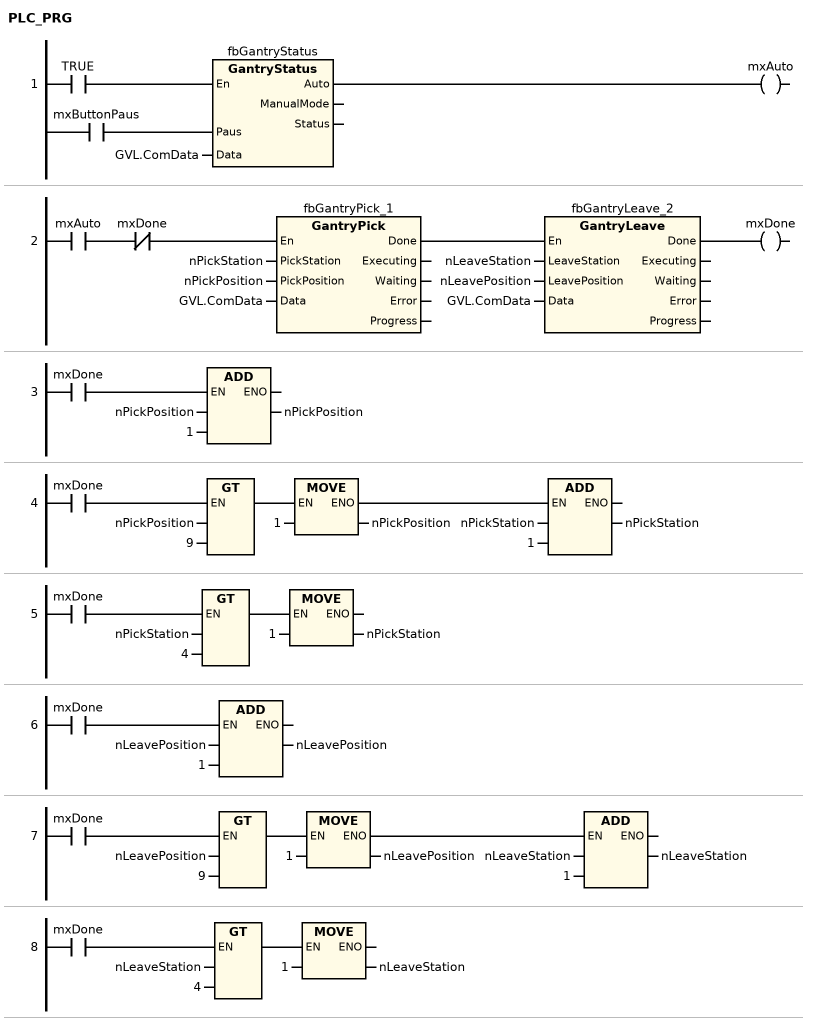
// NETWORK 1
fbGantryStatus(En := TRUE, Paus := mxButtonPaus, Data := GVL.ComData); // GantryStatus
mxAuto := fbGantryStatus.Auto;

// NETWORK 2
fbGantryPick_1(
    En := mxAuto AND NOT mxDone,
    PickStation := nPickStation,
    PickPosition := nPickPosition,
    Data := GVL.ComData); // GantryPick
fbGantryLeave_2(
    En := fbGantryPick_1.Done,
    LeaveStation := nLeaveStation,
    LeavePosition := nLeavePosition,
    Data := GVL.ComData); // GantryLeave
mxDone := fbGantryLeave_2.Done;

// NETWORK 3
IF mxDone THEN nPickPosition := nPickPosition + 1; END_IF

// NETWORK 4
_w1 := mxDone AND nPickPosition > 9;
IF _w1 THEN nPickPosition := 1; END_IF
IF _w1 THEN nPickStation := nPickStation + 1; END_IF

// NETWORK 5
IF mxDone AND nPickStation > 4 THEN nPickStation := 1; END_IF

// NETWORK 6
IF mxDone THEN nLeavePosition := nLeavePosition + 1; END_IF

// NETWORK 7
_w2 := mxDone AND nLeavePosition > 9;
IF _w2 THEN nLeavePosition := 1; END_IF
IF _w2 THEN nLeaveStation := nLeaveStation + 1; END_IF

// NETWORK 8
IF mxDone AND nLeaveStation > 4 THEN nLeaveStation := 1; END_IF

END_PROGRAM

// ---- POUs/GantryStatus.TcPOU
FUNCTION_BLOCK GantryStatus
VAR_INPUT
	En: BOOL;	
	Paus: BOOL;
END_VAR
VAR_OUTPUT
	Auto : BOOL;
	ManualMode : BOOL;	
	Status : STRING;
END_VAR
VAR_IN_OUT
	Data:CommunicationData;
END_VAR
VAR
	fbTonStartDelay: TON;
END_VAR


fbTonStartDelay( IN := Data.Auto, PT := T#1S);


Auto 		:= fbTonStartDelay.Q;
ManualMode 	:= Data.ManualMode;
Status 		:= Data.Status;
Data.Paus := Paus;

END_FUNCTION_BLOCK

// ---- POUs/GantryPick.TcPOU
FUNCTION_BLOCK GantryPick
VAR_INPUT
	En: BOOL;
	PickStation: INT;
	PickPosition: INT;
END_VAR
VAR_OUTPUT
	Done: BOOL;
	Executing: BOOL;
	Waiting: BOOL;
	Error: BOOL;
	Progress: INT;
END_VAR
VAR_IN_OUT
	Data:CommunicationData;
END_VAR
VAR
END_VAR


IF En THEN

	// Auto sequence pick pallet
	CASE Progress OF
		0:	//Clear old order
			Data.PickStation := 0;
			Data.PickPosition := 0;
			Progress := 10;

		10:	//Start gantry robot auto squence
			IF Data.Auto AND PickStation > 0 AND  PickStation <= 4 AND PickPosition > 0 AND PickPosition <= 9 THEN
				Data.PickStation := PickStation;
				Data.PickPosition := PickPosition;
				Executing := FALSE;
				Waiting := FALSE;
				Error := FALSE;
				Progress := 30;
			ELSE
				Executing := FALSE;
				Waiting := FALSE;
				Error := TRUE;
			END_IF

		30: // Check acknowledge from GantryRobot
			IF Data.AckPickStation = PickStation AND Data.AckPickPosition = PickPosition THEN
				Executing := TRUE;
				Waiting := FALSE;
				Error := FALSE;
				Progress := 50;
			ELSE
				Executing := FALSE;
				Waiting := TRUE;
				Error := NOT Data.Auto;
			END_IF
			
		50: // Wait for gantry auto squence ready and clear order	
			IF Data.AckPickStation = 0 AND Data.AckPickPosition = 0 THEN
				Data.PickStation := 0;
				Data.PickPosition := 0;
				Executing := FALSE;
				Waiting := FALSE;
				Error := FALSE;
				Progress := 100;
			ELSE
				Executing := TRUE;
				Waiting := FALSE;
				Error := NOT Data.Auto;
			END_IF
		
		100: // Operation done
			Done := TRUE;
	END_CASE

ELSE //En
	IF Progress > 0 THEN
		Data.PickStation := 0;
		Data.PickPosition := 0;	
	END_IF
	Progress := 0;
	Done := FALSE;
	Executing := FALSE;
	Waiting := FALSE;
	Error := FALSE;
END_IF

END_FUNCTION_BLOCK

// ---- POUs/GantryLeave.TcPOU
FUNCTION_BLOCK GantryLeave
VAR_INPUT
	En: BOOL;
	LeaveStation: INT;
	LeavePosition: INT;
END_VAR
VAR_OUTPUT
	Done: BOOL;
	Executing: BOOL;
	Waiting: BOOL;
	Error: BOOL;
	Progress: INT;
END_VAR
VAR_IN_OUT
	Data:CommunicationData;
END_VAR
VAR
END_VAR

IF En THEN
	
	// Auto sequence leave pallet
	CASE Progress OF
		0:	//Clear old order
			Data.LeaveStation := 0;
			Data.LeavePosition := 0;
			Progress := 10;

		10:	//Start gantry robot auto squence
			IF Data.Auto AND LeaveStation > 0 AND  LeaveStation <= 4 AND LeavePosition > 0 AND LeavePosition <= 9 THEN
				Data.LeaveStation  := LeaveStation;
				Data.LeavePosition := LeavePosition;
				Executing := FALSE;
				Waiting := FALSE;
				Error := FALSE;
				Progress := 30;
			ELSE
				Executing := FALSE;
				Waiting := FALSE;
				Error := TRUE;
			END_IF

		30: // Check acknowledge from GantryRobot
			IF Data.AckLeaveStation = LeaveStation AND Data.AckLeavePosition = LeavePosition THEN
				Executing := TRUE;
				Waiting := FALSE;
				Error := FALSE;
				Progress := 50;
			ELSE
				Executing := FALSE;
				Waiting := TRUE;
				Error := NOT Data.Auto;
			END_IF
			
		50: // Wait for gantry auto squence ready and clear order	
			IF Data.AckLeaveStation = 0 AND Data.AckLeavePosition = 0 THEN
				Data.LeaveStation := 0;
				Data.LeavePosition := 0;
				Executing := FALSE;
				Waiting := FALSE;
				Error := FALSE;
				Progress := 100;
			ELSE
				Executing := TRUE;
				Waiting := FALSE;
				Error := NOT Data.Auto;
			END_IF
		
		100: // Operation done
			Done := TRUE;
	END_CASE

ELSE //En
	IF Progress > 0 THEN
		Data.LeaveStation := 0;
		Data.LeavePosition := 0;	
	END_IF
	Progress := 0;
	Done := FALSE;
	Executing := FALSE;
	Waiting := FALSE;
	Error := FALSE;
END_IF

END_FUNCTION_BLOCK

// ---- GlobalTextList.TcGTLO
TEXTLIST GlobalTextList
  263 = ' Y-Axis %s'
  1185 = '%s'
  489 = 'ABB Go To Conveyor 1'
  490 = 'ABB Go To Conveyour 2'
  485 = 'ABB Go To Home'
  486 = 'ABB Go To Sensor'
  487 = 'ABB Go To Storage'
  488 = 'ABB Go To Table'
  986 = 'ABB PickLeave Conv. 1'
  987 = 'ABB PickLeave Conv. 2'
  983 = 'ABB PickLeave Sensor'
  984 = 'ABB PickLeave Storage'
  985 = 'ABB PickLeave Table'
  840 = 'ABB Status'
  91 = 'Actual Axes Positions'
  67 = 'Actual Position X-Axis %S'
  780 = 'Actual Position X-Axis %s'
  374 = 'Actual Position Y-Axis %s'
  492 = 'Actual Position Z-Axis %s'
  746 = 'AUTO'
  191 = 'Auto                        Manual'
  126 = 'Auto                  Manual'
  493 = 'Auto: %s'
  762 = 'Auto: %s    mm/s'
  413 = 'Auto: %s mm/s'
  269 = 'Axtual Position X %s'
  686 = 'Black Stop Button'
  694 = 'Busy'
  491 = 'By Pass'
  514 = 'By Pass \nEnd Limit X'
  336 = 'By Pass End Limit'
  214 = 'Calibrate Axes'
  695 = 'Communicator'
  965 = 'Communicator Enable'
  430 = 'Control On'
  1616 = "Don't forget to save changes!"
  1083 = "Don't forget to save!"
  998 = 'Done'
  1640 = 'Dont forget to save Positions'
  137 = 'Dont forget to save the \nPositions!'
  194 = 'Dont forget to save the Positions!'
  473 = 'Edit \nSTN100'
  458 = 'EM Stop'
  992 = 'EM Stop OK'
  724 = 'Emergency Stop'
  624 = 'Emergency Stop OK'
  505 = 'Emergency Stopop OK'
  936 = 'End Limit SW'
  66 = 'End Limit SW '
  765 = 'End Limit SW OK'
  1001 = 'Error'
  696 = 'Error %s'
  999 = 'Executing'
  997 = 'Function call'
  465 = 'Gantry Leave'
  464 = 'Gantry Pick'
  81 = 'Gantry Robot'
  441 = 'Gantry Robot\nMenu'
  566 = 'Gate '
  402 = 'Gate Closed'
  571 = 'Gate Closed and Reset'
  567 = 'Gate Closed and reseted'
  1091 = 'Gate Closed and Reseted'
  788 = 'Gate Closed Reset'
  43 = 'Gate OK '
  109 = 'General Conditions'
  996 = 'General Control '
  210 = 'General Control \nOn'
  174 = 'General Control On'
  60 = 'General Power\nOff'
  708 = 'General Power\nOn'
  404 = 'Go To '
  935 = 'Go To \nPosition'
  4 = 'Go To \nStorage Position'
  443 = 'Go To Storage Position'
  829 = 'Gripper'
  1144 = 'GroupBox'
  605 = 'Heart beat'
  382 = 'HOMING'
  140 = 'Homing X '
  133 = 'Homing Y '
  6 = 'Homing Z'
  543 = 'Light Beam'
  1111 = 'Location: %4.1f'
  729 = 'Location: %S'
  544 = 'Location: %s'
  223 = 'Main Menu'
  74 = 'Manual              Auto'
  621 = 'Manual        Auto'
  468 = 'Manual      Auto'
  459 = 'Manual  LOW Speed'
  595 = 'Manual Controls'
  1043 = 'Manual: %s mm/s'
  362 = 'Mod Pos '
  1483 = 'Mod Pos \n'
  1054 = 'Mod Pos \n\nSelected Location'
  665 = 'Mod Pos \n\nSelected Location'
  246 = 'Mod Pos \nSelected Location'
  692 = 'Modify Storage Position'
  842 = 'Operating mode %d'
  911 = 'Override Speed: %s'
  1219 = 'Override: %s'
  867 = 'Override: %s  %'
  1155 = 'PAUS'
  988 = 'Pick'
  1160 = 'Place'
  783 = 'Place 1'
  284 = 'Place 2'
  781 = 'Place 3'
  250 = 'Place 4'
  703 = 'Place 5'
  343 = 'Place 6'
  1179 = 'Place 7'
  247 = 'Place 8'
  480 = 'Place 9'
  989 = 'Pos\n%s'
  467 = 'Pos \n%s'
  823 = 'Position'
  1392 = 'Position %s'
  946 = 'Power\nOn'
  790 = 'Power \nOff'
  606 = 'Program number: %d'
  330 = 'Read'
  1617 = 'Reference run Axes'
  807 = 'Reset \nServo Drives'
  632 = 'Reset Servo Drives'
  604 = 'RPC Remote Procedural Call'
  603 = 'Running'
  841 = 'Running mode %d'
  1310 = 'SAve'
  1444 = 'Save'
  1220 = 'Save \nPositions!'
  297 = 'Save changes on file!'
  193 = 'Save Ented\nPosition'
  268 = 'Save Entered\nPosition'
  283 = 'Save Entred\nPosition'
  990 = 'Save or Undo changes!'
  1791 = 'Save or UnDo changes!'
  248 = 'Save or UnDo the changes!'
  612 = 'Save or Undo yhe changes!'
  560 = 'Save or UnDo yhe changes!'
  19 = 'Speed Settings'
  101 = 'Start Auto'
  466 = 'Station\n%s'
  945 = 'Station address \n%s'
  396 = 'Station: %S'
  586 = 'Station: %s'
  1075 = 'Status: %s'
  707 = 'STN100'
  226 = 'STN200'
  377 = 'STN300'
  63 = 'STN400'
  625 = 'STN500'
  323 = 'Stop Auto'
  524 = 'Stop Button'
  152 = 'Stop Button (Black)'
  674 = 'Stop Button (Black) OK'
  527 = 'UnDo'
  1089 = 'UnDo Entered'
  363 = 'UnDo Entered \nPosition'
  813 = 'Undo Entered \nPosition'
  1000 = 'Waiting'
  714 = 'X'
  333 = 'X '
  859 = 'X                  Y                Z\nReset\nServo Drives'
  153 = 'X                 Y               Z\nReset\nServo Drives'
  141 = 'X                Y                Z\nReset\nServo Drives'
  436 = 'X                Y               Z\nReset\nServo Drives'
  180 = 'X              Y            Z\nReset\nServo Drives'
  228 = 'X              Y            Z\nReset \nServo Drives'
  327 = 'X              Y            Z\nReset Error\nServo Drives'
  855 = 'X      Y     Z\nReset \nServo Drives'
  289 = 'X +'
  412 = 'X-'
  115 = 'X-Axis %s'
  910 = 'X: %4.1f'
  875 = 'X: %f4.1'
  457 = 'X: %S'
  824 = 'X: %s'
  381 = 'Y'
  482 = 'Y+'
  668 = 'Y-'
  142 = 'Y-Axis %s'
  754 = 'Y: %4.1f'
  879 = 'Y: %f4.1'
  1038 = 'Y: %S'
  245 = 'Y: %s'
  38 = 'z'
  406 = 'Z'
  832 = 'z+'
  975 = 'z-'
  348 = 'Z-Axis %s'
  1274 = 'Z: %4.1f'
  789 = 'Z: %f4.1'
  192 = 'Z: %S'
  655 = 'Z: %s'
END_TEXTLIST

// ---- VISUs/GantryRobotVisu.TcVIS
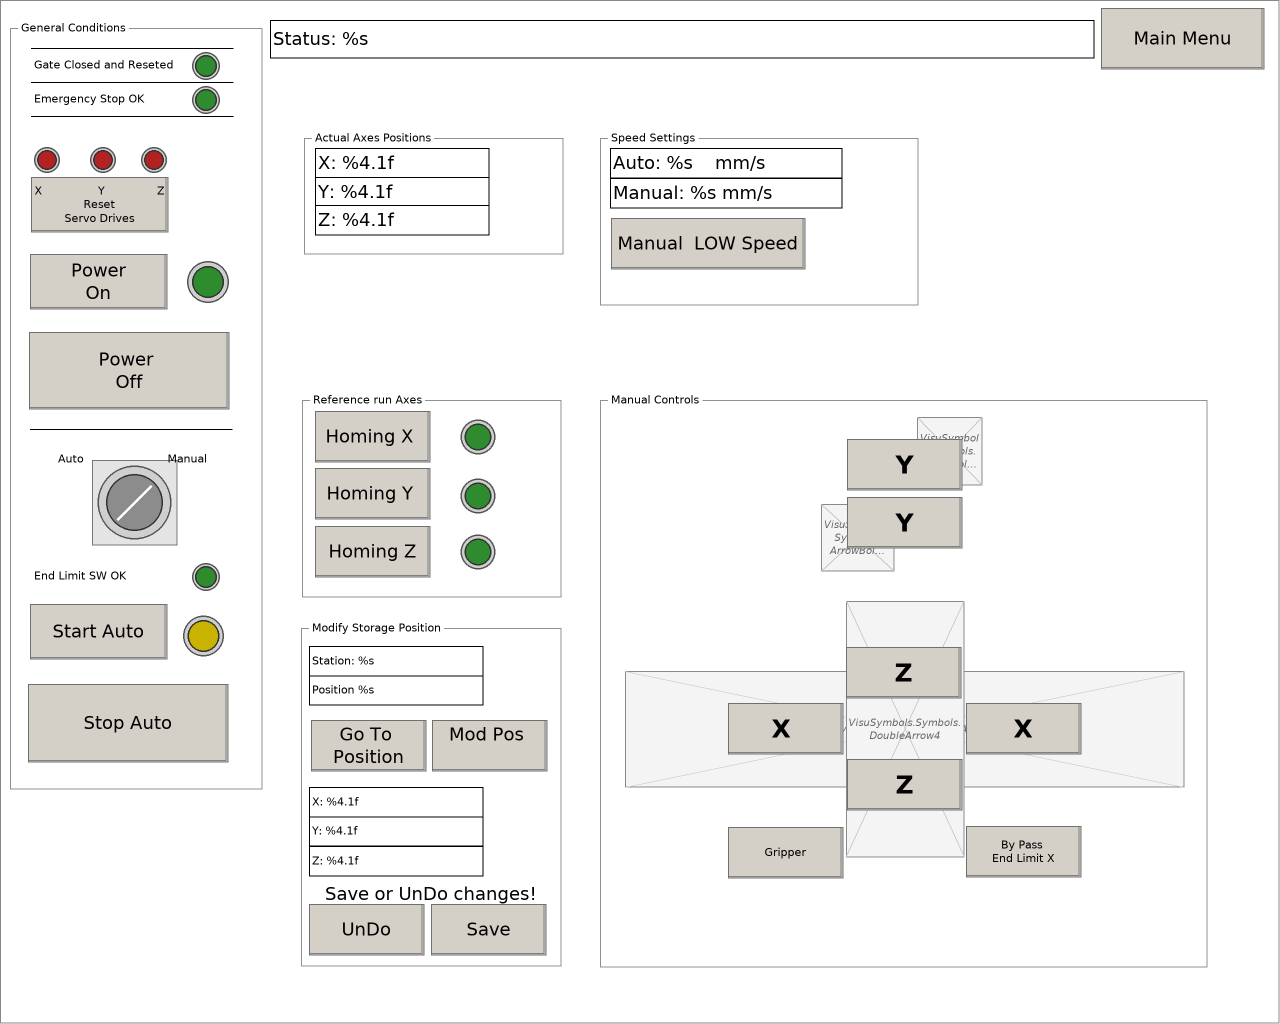
VISUALIZATION GantryRobotVisu  // 1280x1024
    GroupBox (600,392 607x575), "Manual Controls"
        Image (221,112 73x67), image: VisuSymbols.Symbols.ArrowBoldLeftDown
        Image (317,25 65x68), image: VisuSymbols.Symbols.ArrowBoldRightUp
        Image (25,279 559x116), image: VisuSymbols.Symbols.DoubleArrow3
        Image (246,209 118x256), image: VisuSymbols.Symbols.DoubleArrow4
        Button (247,105 115x51), "Y", input disabled if: NOT GantryRobotMotion.mxManualMode
            tap GantryRobotMotion.mxMCYButtonJogFWD
        Button (247,47 115x51), "Y", input disabled if: NOT GantryRobotMotion.mxManualMode
            tap GantryRobotMotion.mxMCYButtonJogBWD
        Button (128,435 115x51), "Gripper", input disabled if: NOT GantryRobotMotion.mxManualMode
            tap GantryRobotMotion.mxTogleGripper
        Button (366,434 115x51), "By Pass End Limit X", invisible if: NOT GantryRobotMotion.mxManualMode, input disabled if: NOT GVL.ixLimSwX
            toggle GantryRobotMotion.mxMCXButtonByPass
        Button (247,367 115x51), "Z", input disabled if: NOT GantryRobotMotion.mxManualMode
            tap GantryRobotMotion.mxMCZButtonJogFWD
        Button (246,255 115x51), "Z", input disabled if: NOT GantryRobotMotion.mxManualMode
            tap GantryRobotMotion.mxMCZButtonJogBWD
        Button (366,311 115x51), "X", input disabled if: NOT GantryRobotMotion.mxManualMode
            tap GantryRobotMotion.mxMCXButtonJogBWD
        Button (128,311 115x51), "X", input disabled if: NOT GantryRobotMotion.mxManualMode
            tap GantryRobotMotion.mxMCXButtonJogFWD
    GroupBox (10,20 252x769), "General Conditions"
        Button (20,234 137x55), "Power On", input disabled if: NOT GantryRobotMotion.mxGeneralCOntrolOk
            tap GantryRobotMotion.mxButtonGeneralControlOn
        Label (21,36 150x32)
        Label (21,29 160x32), "Gate Closed and Reseted"
        Lamp1 (178,30 36x32), variable: GVL.ixLightBeamAndGatesClosed, style: Lamp-Lamp1-Green
        Label (21,63 157x32), "Emergency Stop OK"
        Lamp1 (178,64 36x32), variable: GVL.ixEmergencyStopOk, style: Lamp-Lamp1-Green
        Lamp1 (170,238 56x48), variable: GVL.qxIndControlOn, style: Lamp-Lamp1-Green
        Lamp1 (170,592 47x48), variable: GVL.qxIndProgramStart, style: Lamp-Lamp1-Yellow
        Label (21,540 120x32), "End Limit SW OK"
        Lamp1 (178,541 36x32), variable: GantryRobotMotion.mxLimSwOK, style: Lamp-Lamp1-Green
        Line (21,28) (223,28)
        Line (21,62) (223,62)
        Line (21,96) (223,96)
        RotarySwitch (75,440 99x85), variable: GantryRobotMotion.mxButtonAutoMode, behaviour: TOGGLE, style: Switch-RotarySwitch-Gray
        Label (26,423 193x32), "Auto Manual"
        Line (20,409) (222,409)
        Button (20,584 137x55), "Start Auto", input disabled if: NOT GantryRobotMotion.mxAutoMode
            tap GantryRobotMotion.mxButtonStartAuto
        Lamp1 (128,125 32x30), variable: GantryRobotMotion.mxMCXAxisError, style: Lamp-Lamp1-Red
        Lamp1 (77,125 32x30), variable: GantryRobotMotion.mxMCXAxisError, style: Lamp-Lamp1-Red
        Lamp1 (21,125 32x30), variable: GantryRobotMotion.mxMCXAxisError, style: Lamp-Lamp1-Red
        Button (21,157 137x55), "X Y Z Reset Servo Drives"
            tap GantryRobotMotion.mxButtonResetError
        Button (19,312 200x77), "Power Off", input disabled if: NOT GantryRobotMotion.mxGeneralCOntrolOk
            tap GantryRobotMotion.mxButtonGeneralControlOff
        Button (18,664 200x78), "Stop Auto", input disabled if: NOT GantryRobotMotion.mxAutoMode
            tap GantryRobotMotion.mxButtonStopAuto
    GroupBox (304,130 259x124), "Actual Axes Positions"
        Rectangle (11,18 174x30), "X: %4.1f", text variable: GantryRobotMotion.MCActualPos.x
        Rectangle (11,47 174x30), "Y: %4.1f", text variable: GantryRobotMotion.MCActualPos.y
        Rectangle (11,75 174x30), "Z: %4.1f", text variable: GantryRobotMotion.MCActualPos.z
    Button (1101,8 163x61), "Main Menu"
        OnMouseClick: change screen: Visualization
    Rectangle (270,20 824x38), "Status: %s", text variable: GantryRobotMotion.strStatusText
    GroupBox (600,130 318x175), "Speed Settings"
        Rectangle (10,18 232x30), "Auto: %s mm/s", text variable: GantryRobotMotion.MCAutoVelocity
            OnMouseClick: write the text variable via VisuDialogs.Numpad, min 100, max 1000, title 'Auto Speed mm/s', format %i
        Rectangle (10,48 232x30), "Manual: %s mm/s", text variable: GantryRobotMotion.MCJogVelocity
            OnMouseClick: write the text variable via VisuDialogs.Numpad, min 5, max 250, title 'Jog Speed mm/s', format %i
        Button (11,88 194x51), "Manual LOW Speed", input disabled if: NOT GantryRobotMotion.mxManualMode
            toggle GantryRobotMotion.mxMCButtonManLowVelocity
    GroupBox (301,620 260x346), "Modify Storage Position"
        Button (131,100 115x51), "Mod Pos", input disabled if: NOT GantryRobotMotion.mxManualMode OR NOT GantryRobotMotion.mxHomingDone
            tap GantryRobotMotion.mxButtonModPosExecute
        Rectangle (8,55 174x30), "Position %s", text variable: GantryRobotMotion.ModPosLocation, input disabled if: NOT GantryRobotMotion.mxManualMode
            OnMouseClick: write GantryRobotMotion.ModPosLocation via VisuDialogs.Numpad, min 1, max 9, title "Loacation", format %i
        Button (10,100 115x51), "Go To Position", input disabled if: NOT GantryRobotMotion.mxManualMode OR NOT GantryRobotMotion.mxHomingDone
            tap GantryRobotMotion.mxButtonGoToModPos
        Rectangle (8,26 174x30), "Station: %s", text variable: GantryRobotMotion.ModPosStation, input disabled if: NOT GantryRobotMotion.mxManualMode
            OnMouseClick: write GantryRobotMotion.ModPosStation via VisuDialogs.Numpad, min 1, max 4, title "Station", format %i
        Rectangle (8,196 174x30), "Y: %4.1f", text variable: GantryRobotMotion.arrAbsPosition[GantryRobotMotion.ModPosStation, GantryRobotMotion.ModPosLocation].y, input disabled if: NOT GantryRobotMotion.mxManualMode
            OnMouseClick: write the text variable via VisuDialogs.Numpad, title 'Position Y', format %f
            OnMouseClick: execute { GantryRobotMotion.mxReminderToSave := TRUE; }
        Rectangle (8,226 174x30), "Z: %4.1f", text variable: GantryRobotMotion.arrAbsPosition[GantryRobotMotion.ModPosStation, GantryRobotMotion.ModPosLocation].z, input disabled if: NOT GantryRobotMotion.mxManualMode
            OnMouseClick: write the text variable via VisuDialogs.Numpad, title 'Position Z', format %f
            OnMouseClick: execute { GantryRobotMotion.mxReminderToSave := TRUE; }
        Button (130,284 115x51), "Save", input disabled if: NOT GantryRobotMotion.mxManualMode
            tap GantryRobotMotion.mxButtonSavePos
        Button (8,284 115x51), "UnDo", input disabled if: NOT GantryRobotMotion.mxManualMode
            tap GantryRobotMotion.mxButtonReadFile
        Rectangle (8,167 174x30), "X: %4.1f", text variable: GantryRobotMotion.arrAbsPosition[GantryRobotMotion.ModPosStation, GantryRobotMotion.ModPosLocation].x, input disabled if: NOT GantryRobotMotion.mxManualMode
            OnMouseClick: write the text variable via VisuDialogs.Numpad, title 'Position Z', format %f
            OnMouseClick: execute { GantryRobotMotion.mxReminderToSave := TRUE; }
    GroupBox (302,392 259x205), "Reference run Axes"
        Lamp1 (156,140 40x40), variable: GantryRobotMotion.mxMCZHomingDone, style: Lamp-Lamp1-Green
        Lamp1 (156,84 40x40), variable: GantryRobotMotion.mxMCYHomingDone, style: Lamp-Lamp1-Green
        Lamp1 (156,25 40x40), variable: GantryRobotMotion.mxMCXHomingDone, style: Lamp-Lamp1-Green
        Button (13,134 115x51), "Homing Z", input disabled if: NOT GantryRobotMotion.mxManualMode
            tap GantryRobotMotion.mxMCZButtonHoming
        Button (13,76 115x51), "Homing Y", input disabled if: NOT GantryRobotMotion.mxManualMode
            tap GantryRobotMotion.mxMCYButtonHoming
        Button (13,19 115x51), "Homing X", input disabled if: NOT GantryRobotMotion.mxManualMode
            tap GantryRobotMotion.mxMCXButtonHoming
    Label (306,880 250x28), "Save or UnDo changes!", invisible if: NOT GantryRobotMotion.mxReminderToSave
END_VISUALIZATION

// ---- VISUs/Visualization.TcVIS
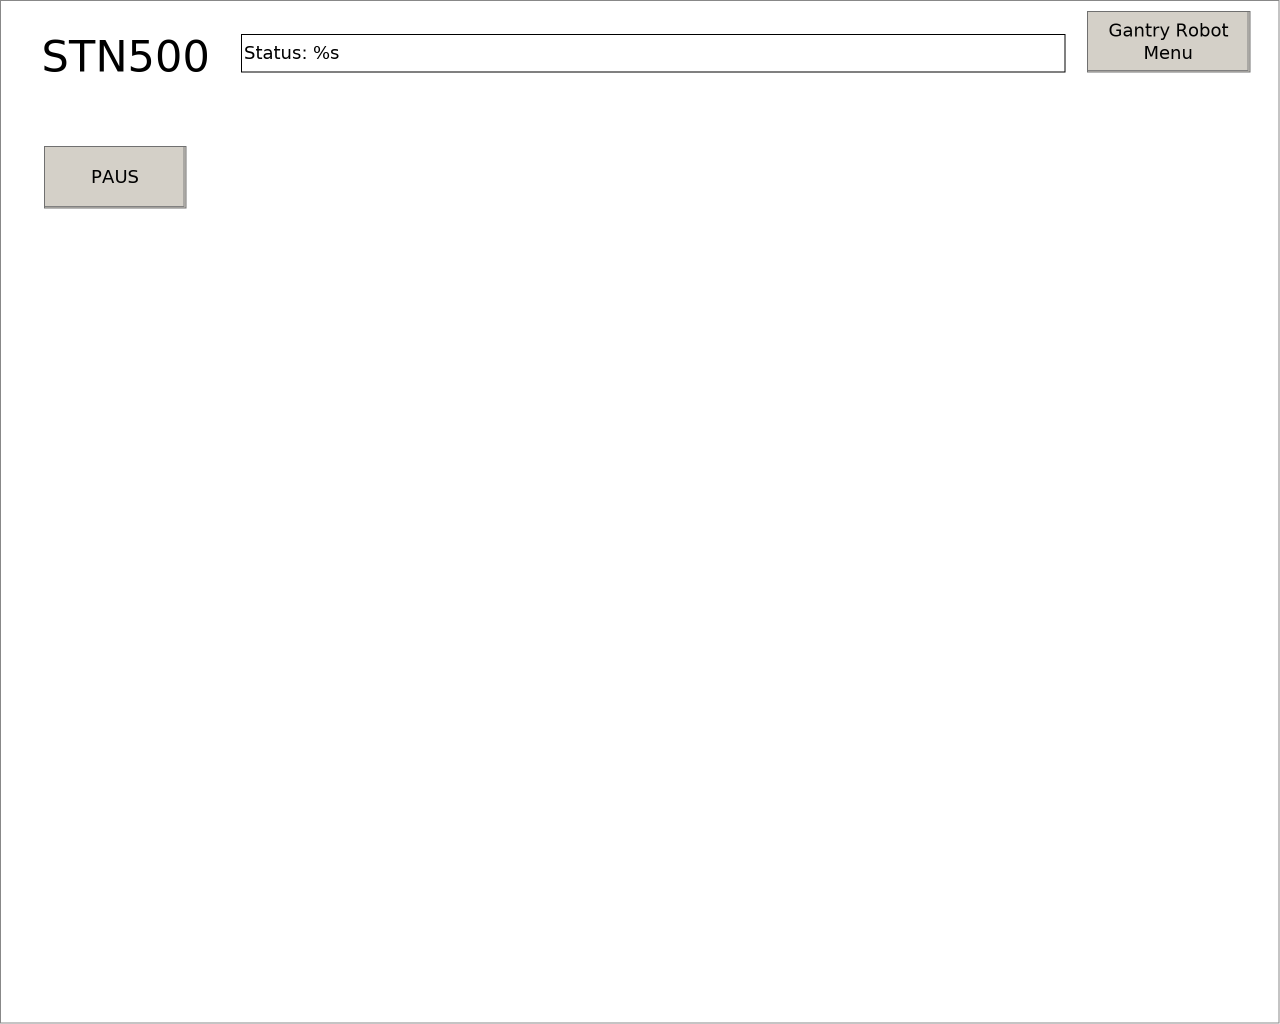
VISUALIZATION Visualization  // 1280x1024
    Label (18,0 216x113), "STN500"
    Button (1087,11 163x61), "Gantry Robot Menu"
        OnMouseClick: change screen: GantryRobotVisu
    Rectangle (241,34 824x38), "Status: %s", text variable: PLC_PRG.fbGantryStatus.Status
    Button (44,146 142x62), "PAUS", input disabled if: NOT PLC_PRG.mxAuto
        toggle PLC_PRG.mxButtonPaus
END_VISUALIZATION
